// TwinCAT 3 PLC project Main_PLC_Project
// ProgramVersion: 3.1.4023.0
// libraries:
//   Tc2_ControllerToolbox, * (Beckhoff Automation GmbH)
//   Tc2_MC2, * (Beckhoff Automation GmbH)
//   Tc2_MC2_Drive, * (Beckhoff Automation GmbH)
//   Tc2_SerialCom, * (Beckhoff Automation GmbH)
//   Tc2_Standard, * (Beckhoff Automation GmbH)
//   Tc2_System, * (Beckhoff Automation GmbH)
//   Tc3_Filter, * (Beckhoff Automation GmbH)
//   Tc3_Module, * (Beckhoff Automation GmbH)
//   TcMatrix,1.3.0,Burks Engineering
// project tree:
//   DUTs/ E_RobotMode.TcDUT, ST_FilterParams.TcDUT, tDataFrame.TcDUT
//   GVLs/ CONSTANTS.TcGVL, Control.TcGVL, HmiToPlc.TcGVL, Parameters.TcGVL, PlcToHmi.TcGVL, RobotParams.TcGVL, Safety.TcGVL
//   IMU/DUTs/ E_FilterOrder.TcDUT, E_SerialError.TcDUT, E_SerialState.TcDUT, ST_ImuData.TcDUT, ST_JointLimits.TcDUT, ST_JointOffsets.TcDUT, ST_JointParameters.TcDUT, ST_Vector3.TcDUT, tDataFrame_1.TcDUT
//   IMU/GVLs/ IMU.TcGVL
//   IMU/POUs/ ATAN2.TcPOU, BackgroundCOM.TcPOU, FB_AccelerometerAngle.TcPOU, FB_ComplementaryFilter.TcPOU, FB_GetSerialData.TcPOU, FB_MapStim300.TcPOU
//   MATRIX/ AccelerometerReadings.TcPOU, FB_Matrix3x3.TcPOU, FB_Matrix4x4.TcPOU, FB_Vector3.TcPOU, F_Cross2.TcPOU, F_DH.TcPOU
//   / PlcTask.TcTTO, SerialComTask.TcTTO
//   POUs/ FB_Joint.TcPOU, FB_Robot3R.TcPOU, FB_LowPassFilter.TcPOU, FB_TorqueController.TcPOU, FB_TrajectoryGenerator.TcPOU, F_Merge24BitSigned.TcPOU, F_Merge24BitUnsigned.TcPOU, MAIN.TcPOU, P_HMI.TcPOU, RescaleRange.TcPOU
// real-time tasks:
//   TASK PlcTask: cycle T#10ms, priority 20, ADS port 350
//   TASK SerialComTask: cycle T#1ms, priority 1, ADS port 351
// motion (NC):
//   TASK Main_NC_Task SAF: cycle T#2ms, priority 4, ADS port 501
//   TASK Main_NC_Task SVB: cycle T#10ms, priority 8, ADS port 511
//   AXIS Axis1_Drive1_Joint1 (id 1)
//     General: UnitName=°
//     Dynamic: AccelerationMaximum=44, DecelerationMaximum=44, Acceleration=229.701756820377, Deceleration=229.701756820377, Jerk=689.10527046113
//     Velo: RefSearch=1.53134504546918, RefSync=1.53134504546918, SlowManual=7.65672522734589, FastManual=45.9403513640753, Fast=153.134504546918, Maximum=153.134504546918
//     OtherSettings: AllowMotionCmdToSlave=true, PulseDistancePos=1, PulseDistanceNeg=1
//     encoder EncType=8
//       EncPara: ScaleFactorNumerator=5.901639, ScaleFactorDenominator=1048576, MaxCount=#xffffffff
//         SoftEndMinControl: Enable=true, Range=-20
//         SoftEndMaxControl: Enable=true, Range=20
//     drive DrvType=9
//       DrvPara: MaxCount=#xffffffff, DriveControlDWord=#x00030000
//         Analog: VeloReferenz=168.44795500161, VeloScale=1.02400649589962, TorqueSetpointScale=10, ScaleFactorActTorque=0.1
//         TimeComp: TaskDelayCycles=1
//     controller CtrType=1
//       CtrPara: PriorControlFactor=1
//         Observer: BandWidth=20
//   AXIS Axis1_Drive2_Joint2 (id 3)
//     General: UnitName=°
//     Dynamic: AccelerationMaximum=76, DecelerationMaximum=76, Acceleration=389.12958984375, Deceleration=389.12958984375, Jerk=1167.38876953125
//     Velo: RefSearch=2.594197265625, RefSync=2.594197265625, SlowManual=12.970986328125, FastManual=77.82591796875, Fast=259.4197265625, Maximum=259.4197265625
//     OtherSettings: AllowMotionCmdToSlave=true, PulseDistancePos=1, PulseDistanceNeg=1
//     encoder EncType=8
//       EncPara: ScaleFactorNumerator=7.2, ScaleFactorDenominator=1048576, MaxCount=#xffffffff
//         SoftEndMinControl: Enable=true, Range=-95
//         SoftEndMaxControl: Enable=true, Range=95
//     drive DrvType=9
//       DrvPara: MaxCount=#xffffffff, DriveControlDWord=#x00030000
//         Analog: VeloReferenz=285.36169921875, VeloScale=1.02400649589962, TorqueSetpointScale=10, ScaleFactorActTorque=0.1
//         TimeComp: TaskDelayCycles=1
//     controller CtrType=1
//       CtrPara: PriorControlFactor=1
//         Observer: BandWidth=20
//   AXIS Axis1_Drive3_Joint3 (id 5)
//     General: UnitName=Degree
//     Dynamic: AccelerationMaximum=865.888117688623, DecelerationMaximum=865.888117688623, Acceleration=865.888, Deceleration=865.888, Jerk=2597.66, OverrideType=4
//     Velo: RefSearch=5.77258745125749, RefSync=5.77258745125749, SlowManual=28.8629372562874, FastManual=173.177623537725, Fast=577.258745125749, Maximum=577.259
//     OtherSettings: AllowMotionCmdToSlave=true, PulseDistancePos=1, PulseDistanceNeg=1
//     encoder EncType=8
//       EncPara: ScaleFactorNumerator=10.285714, ScaleFactorDenominator=1048576, MaxCount=#xffffffff
//         SoftEndMinControl: Enable=true, Range=-95
//         SoftEndMaxControl: Enable=true, Range=95
//     drive DrvType=9
//       DrvPara: MaxCount=#xffffffff, DriveControlDWord=#x00030000
//         Analog: VeloReferenz=634.984619638324, VeloScale=1.02400649589962, TorqueSetpointScale=10, ScaleFactorActTorque=0.1
//         TimeComp: TaskDelayCycles=1
//     controller CtrType=1
//       CtrPara: PriorControlFactor=1
//         PID: PosTv=0.5, PosTd=0.1, VeloTv=0.2, VeloTd=0.08
//         Observer: BandWidth=20
// I/O:
//   DEVICE Device 5 (EtherCAT), AmsNetId 5.72.215.242.6.1
//     Drive1_Joint1 (AX5106-0000-0210) [AX5106-0000-0210 EtherCAT Drive (SoE, 1 Ch.)]
//       Term 10 (AX5805) [AX5805 (Safety Drive Option)]
//         modules: Module 1 (Safety Process Data, 1 axis), Module 2 (Standard Process Data, 1 axis)
//       Term 7 (EL9011) [EL9011 End Terminal]
//     Drive2_Joint2(AX5106-0000-0210) [AX5106-0000-0210 EtherCAT Drive (SoE, 1 Ch.)]
//       Term 11 (AX5805) [AX5805 (Safety Drive Option)]
//         modules: Module 1 (Safety Process Data, 1 axis), Module 2 (Standard Process Data, 1 axis)
//       Term 8 (EL9011) [EL9011 End Terminal]
//     Drive3_Joint3(AX5106-0000-0210) [AX5106-0000-0210 EtherCAT Drive (SoE, 1 Ch.)]
//       Term 12 (AX5805) [AX5805 (Safety Drive Option)]
//         modules: Module 1 (Safety Process Data, 1 axis), Module 2 (Standard Process Data, 1 axis)
//       Term 9 (EL9011) [EL9011 End Terminal]
//     Box 22 (Leica-RT-Output) [Leica RT Output] (disabled)
//   DEVICE Device 1 (EtherCAT), AmsNetId 5.72.215.242.2.1
//     Term 5 (EK1200) [EK1200-5000 EtherCAT Power supply (2A E-Bus)]
//       Term 14 (EL6900) [EL6900, TwinSAFE PLC]
//       Term 15 (EL1904) [EL1904, 4 Ch. Safety Input 24V, TwinSAFE]
//         modules: Module 1 (FSOES)
//       Term 16 (EL6022) [EL6022 Interface 2Ch. (RS422/485)]
//       Term 19 (EL6022) [EL6022 Interface 2Ch. (RS422/485)]
//       Term 9 (EL9011) [EL9011 End Terminal]
// variable links:
//   Device 1 (EtherCAT) <-> Device 1 (EtherCAT)/Term 5 (EK1200)/Term 14 (EL6900)
//     Term 5 (EK1200)/Term 15 (EL1904)/Module 1 (FSOES)/RxPDO/FSOE <-> ConnectionInputs/Message_9 TxPDO
//     Term 5 (EK1200)/Term 15 (EL1904)/Module 1 (FSOES)/TxPDO/FSOE <-> ConnectionOutputs/Message_9 RxPDO
//   Device 1 (EtherCAT) <-> Device 5 (EtherCAT)/Drive1_Joint1 (AX5106-0000-0210)/Term 10 (AX5805)
//     Term 5 (EK1200)/Term 14 (EL6900)/ConnectionOutputs/Message_6 RxPDO <-> Module 1 (Safety Process Data, 1 axis)/Inputs (Statusword)/FSOE
//   Device 5 (EtherCAT) <-> Device 1 (EtherCAT)/Term 5 (EK1200)/Term 14 (EL6900)
//     Drive1_Joint1 (AX5106-0000-0210)/Term 10 (AX5805)/Module 1 (Safety Process Data, 1 axis)/Outputs (Controlword)/FSOE <-> ConnectionInputs/Message_6 TxPDO
//     Drive2_Joint2(AX5106-0000-0210)/Term 11 (AX5805)/Module 1 (Safety Process Data, 1 axis)/Inputs (Statusword)/FSOE <-> ConnectionOutputs/Message_7 RxPDO
//     Drive3_Joint3(AX5106-0000-0210)/Term 12 (AX5805)/Module 1 (Safety Process Data, 1 axis)/Inputs (Statusword)/FSOE <-> ConnectionOutputs/Message_8 RxPDO
//     Drive2_Joint2(AX5106-0000-0210)/Term 11 (AX5805)/Module 1 (Safety Process Data, 1 axis)/Outputs (Controlword)/FSOE <-> ConnectionInputs/Message_7 TxPDO
//     Drive3_Joint3(AX5106-0000-0210)/Term 12 (AX5805)/Module 1 (Safety Process Data, 1 axis)/Outputs (Controlword)/FSOE <-> ConnectionInputs/Message_8 TxPDO
//   Main_NC_Task SAF/Axes/Axis1_Drive1_Joint1 <-> Device 5 (EtherCAT)/Drive1_Joint1 (AX5106-0000-0210)
//     Drive/Inputs/In/nDcOutputTime <-> InfoData/DcOutputShift
//     Drive/Inputs/In/nState1 <-> AT/Drive status word @bit 8
//     Drive/Inputs/In/nState2 <-> AT/Drive status word
//     Drive/Inputs/In/nState4 @bit 1 <-> WcState/InputToggle
//     Drive/Inputs/In/nState4 <-> WcState/WcState
//     Drive/Outputs/Out/nCtrl1 <-> MDT/Master control word @bit 8
//     Drive/Outputs/Out/nDataOut2 <-> MDT/Velocity command value
//     Enc/Inputs/In/nDataIn1 <-> AT/Position feedback 1 value (motor feedback)
//     Enc/Inputs/In/nDcInputTime <-> InfoData/DcInputShift
//     Enc/Inputs/In/nState4 @bit 1 <-> WcState/InputToggle
//     Enc/Inputs/In/nState4 <-> WcState/WcState
//   Main_NC_Task SAF/Axes/Axis1_Drive2_Joint2 <-> Device 5 (EtherCAT)/Drive2_Joint2(AX5106-0000-0210)
//     Drive/Inputs/In/nDcOutputTime <-> InfoData/DcOutputShift
//     Drive/Inputs/In/nState1 <-> AT/Drive status word @bit 8
//     Drive/Inputs/In/nState2 <-> AT/Drive status word
//     Drive/Inputs/In/nState4 @bit 1 <-> WcState/InputToggle
//     Drive/Inputs/In/nState4 <-> WcState/WcState
//     Drive/Outputs/Out/nCtrl1 <-> MDT/Master control word @bit 8
//     Drive/Outputs/Out/nDataOut2 <-> MDT/Velocity command value
//     Enc/Inputs/In/nDataIn1 <-> AT/Position feedback 1 value (motor feedback)
//     Enc/Inputs/In/nDcInputTime <-> InfoData/DcInputShift
//     Enc/Inputs/In/nState4 @bit 1 <-> WcState/InputToggle
//     Enc/Inputs/In/nState4 <-> WcState/WcState
//   Main_NC_Task SAF/Axes/Axis1_Drive3_Joint3 <-> Device 5 (EtherCAT)/Drive3_Joint3(AX5106-0000-0210)
//     Drive/Inputs/In/nDcOutputTime <-> InfoData/DcOutputShift
//     Drive/Inputs/In/nState1 <-> AT/Drive status word @bit 8
//     Drive/Inputs/In/nState2 <-> AT/Drive status word
//     Drive/Inputs/In/nState4 @bit 1 <-> WcState/InputToggle
//     Drive/Inputs/In/nState4 <-> WcState/WcState
//     Drive/Outputs/Out/nCtrl1 <-> MDT/Master control word @bit 8
//     Drive/Outputs/Out/nDataOut2 <-> MDT/Velocity command value
//     Drive/Outputs/Out/nDataOut4[0] <-> MDT/Torque/force command value
//     Enc/Inputs/In/nDataIn1 <-> AT/Position feedback 1 value (motor feedback)
//     Enc/Inputs/In/nDcInputTime <-> InfoData/DcInputShift
//     Enc/Inputs/In/nState4 @bit 1 <-> WcState/InputToggle
//     Enc/Inputs/In/nState4 <-> WcState/WcState
//   Main_PLC_Project/Main_PLC_Project Instance <-> Device 1 (EtherCAT)/Term 5 (EK1200)/Term 14 (EL6900)
//     PlcTask Inputs/Safety.TS_I_Safety_EStopError <-> StandardInputs/Standard Out Var 5
//     PlcTask Inputs/Safety.TS_I_Safety_EStopOK <-> StandardInputs/Standard Out Var 4
//     PlcTask Outputs/Safety.TS_Q_Safety_Drive_Axis_ErrReset <-> StandardOutputs/Standard In Var 11
//     PlcTask Outputs/Safety.TS_Q_Safety_EStopRestart <-> StandardOutputs/Standard In Var 2
//     PlcTask Outputs/Safety.TS_Q_Safety_GroupPort_ErrAck <-> StandardOutputs/Standard In Var 1
//     PlcTask Outputs/Safety.TS_Q_Safety_GroupPort_RunStop <-> StandardOutputs/Standard In Var 3
//   Main_PLC_Project/Main_PLC_Project Instance <-> Device 1 (EtherCAT)/Term 5 (EK1200)/Term 16 (EL6022)
//     SerialComTask Inputs/IMU.fbStim300[0].stIn_EL6022 @bit 16 <-> COM Inputs Channel 1/Data In 0
//     SerialComTask Inputs/IMU.fbStim300[0].stIn_EL6022 @bit 24 <-> COM Inputs Channel 1/Data In 1
//     SerialComTask Inputs/IMU.fbStim300[0].stIn_EL6022 @bit 96 <-> COM Inputs Channel 1/Data In 10
//     SerialComTask Inputs/IMU.fbStim300[0].stIn_EL6022 @bit 104 <-> COM Inputs Channel 1/Data In 11
//     SerialComTask Inputs/IMU.fbStim300[0].stIn_EL6022 @bit 112 <-> COM Inputs Channel 1/Data In 12
//     SerialComTask Inputs/IMU.fbStim300[0].stIn_EL6022 @bit 120 <-> COM Inputs Channel 1/Data In 13
//     SerialComTask Inputs/IMU.fbStim300[0].stIn_EL6022 @bit 128 <-> COM Inputs Channel 1/Data In 14
//     SerialComTask Inputs/IMU.fbStim300[0].stIn_EL6022 @bit 136 <-> COM Inputs Channel 1/Data In 15
//     SerialComTask Inputs/IMU.fbStim300[0].stIn_EL6022 @bit 144 <-> COM Inputs Channel 1/Data In 16
//     SerialComTask Inputs/IMU.fbStim300[0].stIn_EL6022 @bit 152 <-> COM Inputs Channel 1/Data In 17
//     SerialComTask Inputs/IMU.fbStim300[0].stIn_EL6022 @bit 160 <-> COM Inputs Channel 1/Data In 18
//     SerialComTask Inputs/IMU.fbStim300[0].stIn_EL6022 @bit 168 <-> COM Inputs Channel 1/Data In 19
//     SerialComTask Inputs/IMU.fbStim300[0].stIn_EL6022 @bit 32 <-> COM Inputs Channel 1/Data In 2
//     SerialComTask Inputs/IMU.fbStim300[0].stIn_EL6022 @bit 176 <-> COM Inputs Channel 1/Data In 20
//     SerialComTask Inputs/IMU.fbStim300[0].stIn_EL6022 @bit 184 <-> COM Inputs Channel 1/Data In 21
//     SerialComTask Inputs/IMU.fbStim300[0].stIn_EL6022 @bit 40 <-> COM Inputs Channel 1/Data In 3
//     SerialComTask Inputs/IMU.fbStim300[0].stIn_EL6022 @bit 48 <-> COM Inputs Channel 1/Data In 4
//     SerialComTask Inputs/IMU.fbStim300[0].stIn_EL6022 @bit 56 <-> COM Inputs Channel 1/Data In 5
//     SerialComTask Inputs/IMU.fbStim300[0].stIn_EL6022 @bit 64 <-> COM Inputs Channel 1/Data In 6
//     SerialComTask Inputs/IMU.fbStim300[0].stIn_EL6022 @bit 72 <-> COM Inputs Channel 1/Data In 7
//     SerialComTask Inputs/IMU.fbStim300[0].stIn_EL6022 @bit 80 <-> COM Inputs Channel 1/Data In 8
//     SerialComTask Inputs/IMU.fbStim300[0].stIn_EL6022 @bit 88 <-> COM Inputs Channel 1/Data In 9
//     SerialComTask Inputs/IMU.fbStim300[1].stIn_EL6022 @bit 16 <-> COM Inputs Channel 2/Data In 0
//     SerialComTask Inputs/IMU.fbStim300[1].stIn_EL6022 @bit 24 <-> COM Inputs Channel 2/Data In 1
//     SerialComTask Inputs/IMU.fbStim300[1].stIn_EL6022 @bit 96 <-> COM Inputs Channel 2/Data In 10
//     SerialComTask Inputs/IMU.fbStim300[1].stIn_EL6022 @bit 104 <-> COM Inputs Channel 2/Data In 11
//     SerialComTask Inputs/IMU.fbStim300[1].stIn_EL6022 @bit 112 <-> COM Inputs Channel 2/Data In 12
//     SerialComTask Inputs/IMU.fbStim300[1].stIn_EL6022 @bit 120 <-> COM Inputs Channel 2/Data In 13
//     SerialComTask Inputs/IMU.fbStim300[1].stIn_EL6022 @bit 128 <-> COM Inputs Channel 2/Data In 14
//     SerialComTask Inputs/IMU.fbStim300[1].stIn_EL6022 @bit 136 <-> COM Inputs Channel 2/Data In 15
//     SerialComTask Inputs/IMU.fbStim300[1].stIn_EL6022 @bit 144 <-> COM Inputs Channel 2/Data In 16
//     SerialComTask Inputs/IMU.fbStim300[1].stIn_EL6022 @bit 152 <-> COM Inputs Channel 2/Data In 17
//     SerialComTask Inputs/IMU.fbStim300[1].stIn_EL6022 @bit 160 <-> COM Inputs Channel 2/Data In 18
//     SerialComTask Inputs/IMU.fbStim300[1].stIn_EL6022 @bit 168 <-> COM Inputs Channel 2/Data In 19
//     SerialComTask Inputs/IMU.fbStim300[1].stIn_EL6022 @bit 32 <-> COM Inputs Channel 2/Data In 2
//     SerialComTask Inputs/IMU.fbStim300[1].stIn_EL6022 @bit 176 <-> COM Inputs Channel 2/Data In 20
//     SerialComTask Inputs/IMU.fbStim300[1].stIn_EL6022 @bit 184 <-> COM Inputs Channel 2/Data In 21
//     SerialComTask Inputs/IMU.fbStim300[1].stIn_EL6022 @bit 40 <-> COM Inputs Channel 2/Data In 3
//     SerialComTask Inputs/IMU.fbStim300[1].stIn_EL6022 @bit 48 <-> COM Inputs Channel 2/Data In 4
//     SerialComTask Inputs/IMU.fbStim300[1].stIn_EL6022 @bit 56 <-> COM Inputs Channel 2/Data In 5
//     SerialComTask Inputs/IMU.fbStim300[1].stIn_EL6022 @bit 64 <-> COM Inputs Channel 2/Data In 6
//     SerialComTask Inputs/IMU.fbStim300[1].stIn_EL6022 @bit 72 <-> COM Inputs Channel 2/Data In 7
//     SerialComTask Inputs/IMU.fbStim300[1].stIn_EL6022 @bit 80 <-> COM Inputs Channel 2/Data In 8
//     SerialComTask Inputs/IMU.fbStim300[1].stIn_EL6022 @bit 88 <-> COM Inputs Channel 2/Data In 9
//     SerialComTask Inputs/IMU.fbStim300[0].stIn_EL6022 <-> COM Inputs Channel 1/Status
//     SerialComTask Inputs/IMU.fbStim300[1].stIn_EL6022 <-> COM Inputs Channel 2/Status
//     SerialComTask Outputs/IMU.fbStim300[0].stOut_EL6022 <-> COM Outputs Channel 1/Ctrl
//     SerialComTask Outputs/IMU.fbStim300[1].stOut_EL6022 <-> COM Outputs Channel 2/Ctrl
//     SerialComTask Outputs/IMU.fbStim300[0].stOut_EL6022 @bit 16 <-> COM Outputs Channel 1/Data Out 0
//     SerialComTask Outputs/IMU.fbStim300[0].stOut_EL6022 @bit 24 <-> COM Outputs Channel 1/Data Out 1
//     SerialComTask Outputs/IMU.fbStim300[0].stOut_EL6022 @bit 96 <-> COM Outputs Channel 1/Data Out 10
//     SerialComTask Outputs/IMU.fbStim300[0].stOut_EL6022 @bit 104 <-> COM Outputs Channel 1/Data Out 11
//     SerialComTask Outputs/IMU.fbStim300[0].stOut_EL6022 @bit 112 <-> COM Outputs Channel 1/Data Out 12
//     SerialComTask Outputs/IMU.fbStim300[0].stOut_EL6022 @bit 120 <-> COM Outputs Channel 1/Data Out 13
//     SerialComTask Outputs/IMU.fbStim300[0].stOut_EL6022 @bit 128 <-> COM Outputs Channel 1/Data Out 14
//     SerialComTask Outputs/IMU.fbStim300[0].stOut_EL6022 @bit 136 <-> COM Outputs Channel 1/Data Out 15
//     SerialComTask Outputs/IMU.fbStim300[0].stOut_EL6022 @bit 144 <-> COM Outputs Channel 1/Data Out 16
//     SerialComTask Outputs/IMU.fbStim300[0].stOut_EL6022 @bit 152 <-> COM Outputs Channel 1/Data Out 17
//     SerialComTask Outputs/IMU.fbStim300[0].stOut_EL6022 @bit 160 <-> COM Outputs Channel 1/Data Out 18
//     SerialComTask Outputs/IMU.fbStim300[0].stOut_EL6022 @bit 168 <-> COM Outputs Channel 1/Data Out 19
//     SerialComTask Outputs/IMU.fbStim300[0].stOut_EL6022 @bit 32 <-> COM Outputs Channel 1/Data Out 2
//     SerialComTask Outputs/IMU.fbStim300[0].stOut_EL6022 @bit 176 <-> COM Outputs Channel 1/Data Out 20
//     SerialComTask Outputs/IMU.fbStim300[0].stOut_EL6022 @bit 184 <-> COM Outputs Channel 1/Data Out 21
//     SerialComTask Outputs/IMU.fbStim300[0].stOut_EL6022 @bit 40 <-> COM Outputs Channel 1/Data Out 3
//     SerialComTask Outputs/IMU.fbStim300[0].stOut_EL6022 @bit 48 <-> COM Outputs Channel 1/Data Out 4
//     SerialComTask Outputs/IMU.fbStim300[0].stOut_EL6022 @bit 56 <-> COM Outputs Channel 1/Data Out 5
//     SerialComTask Outputs/IMU.fbStim300[0].stOut_EL6022 @bit 64 <-> COM Outputs Channel 1/Data Out 6
//     SerialComTask Outputs/IMU.fbStim300[0].stOut_EL6022 @bit 72 <-> COM Outputs Channel 1/Data Out 7
//     SerialComTask Outputs/IMU.fbStim300[0].stOut_EL6022 @bit 80 <-> COM Outputs Channel 1/Data Out 8
//     SerialComTask Outputs/IMU.fbStim300[0].stOut_EL6022 @bit 88 <-> COM Outputs Channel 1/Data Out 9
//     SerialComTask Outputs/IMU.fbStim300[1].stOut_EL6022 @bit 16 <-> COM Outputs Channel 2/Data Out 0
//     SerialComTask Outputs/IMU.fbStim300[1].stOut_EL6022 @bit 24 <-> COM Outputs Channel 2/Data Out 1
//     SerialComTask Outputs/IMU.fbStim300[1].stOut_EL6022 @bit 96 <-> COM Outputs Channel 2/Data Out 10
//     SerialComTask Outputs/IMU.fbStim300[1].stOut_EL6022 @bit 104 <-> COM Outputs Channel 2/Data Out 11
//     SerialComTask Outputs/IMU.fbStim300[1].stOut_EL6022 @bit 112 <-> COM Outputs Channel 2/Data Out 12
//     SerialComTask Outputs/IMU.fbStim300[1].stOut_EL6022 @bit 120 <-> COM Outputs Channel 2/Data Out 13
//     SerialComTask Outputs/IMU.fbStim300[1].stOut_EL6022 @bit 128 <-> COM Outputs Channel 2/Data Out 14
//     SerialComTask Outputs/IMU.fbStim300[1].stOut_EL6022 @bit 136 <-> COM Outputs Channel 2/Data Out 15
//     SerialComTask Outputs/IMU.fbStim300[1].stOut_EL6022 @bit 144 <-> COM Outputs Channel 2/Data Out 16
//     SerialComTask Outputs/IMU.fbStim300[1].stOut_EL6022 @bit 152 <-> COM Outputs Channel 2/Data Out 17
//     SerialComTask Outputs/IMU.fbStim300[1].stOut_EL6022 @bit 160 <-> COM Outputs Channel 2/Data Out 18
//     SerialComTask Outputs/IMU.fbStim300[1].stOut_EL6022 @bit 168 <-> COM Outputs Channel 2/Data Out 19
//     SerialComTask Outputs/IMU.fbStim300[1].stOut_EL6022 @bit 32 <-> COM Outputs Channel 2/Data Out 2
//     SerialComTask Outputs/IMU.fbStim300[1].stOut_EL6022 @bit 176 <-> COM Outputs Channel 2/Data Out 20
//     SerialComTask Outputs/IMU.fbStim300[1].stOut_EL6022 @bit 184 <-> COM Outputs Channel 2/Data Out 21
//     SerialComTask Outputs/IMU.fbStim300[1].stOut_EL6022 @bit 40 <-> COM Outputs Channel 2/Data Out 3
//     SerialComTask Outputs/IMU.fbStim300[1].stOut_EL6022 @bit 48 <-> COM Outputs Channel 2/Data Out 4
//     SerialComTask Outputs/IMU.fbStim300[1].stOut_EL6022 @bit 56 <-> COM Outputs Channel 2/Data Out 5
//     SerialComTask Outputs/IMU.fbStim300[1].stOut_EL6022 @bit 64 <-> COM Outputs Channel 2/Data Out 6
//     SerialComTask Outputs/IMU.fbStim300[1].stOut_EL6022 @bit 72 <-> COM Outputs Channel 2/Data Out 7
//     SerialComTask Outputs/IMU.fbStim300[1].stOut_EL6022 @bit 80 <-> COM Outputs Channel 2/Data Out 8
//     SerialComTask Outputs/IMU.fbStim300[1].stOut_EL6022 @bit 88 <-> COM Outputs Channel 2/Data Out 9
//   Main_PLC_Project/Main_PLC_Project Instance <-> Device 1 (EtherCAT)/Term 5 (EK1200)/Term 19 (EL6022)
//     SerialComTask Inputs/IMU.fbStim300[2].stIn_EL6022 @bit {16..184 step 8} <-> COM Inputs Channel 1/Data In {0..21}  (22 links)
//     SerialComTask Inputs/IMU.fbStim300[2].stIn_EL6022 <-> COM Inputs Channel 1/Status
//     SerialComTask Outputs/IMU.fbStim300[2].stOut_EL6022 <-> COM Outputs Channel 1/Ctrl
//     SerialComTask Outputs/IMU.fbStim300[2].stOut_EL6022 @bit {16..184 step 8} <-> COM Outputs Channel 1/Data Out {0..21}  (22 links)
//   Main_PLC_Project/Main_PLC_Project Instance <-> Device 5 (EtherCAT)/Box 22 (Leica-RT-Output)
//     PlcTask Inputs/MAIN.fLeicaRawD <-> Cyclic Measurements/Distance
//     PlcTask Inputs/MAIN.fLeicaRawH <-> Cyclic Measurements/AngleHz
//     PlcTask Inputs/MAIN.fLeicaRawV <-> Cyclic Measurements/AngleVt
//   Main_PLC_Project/Main_PLC_Project Instance <-> Device 5 (EtherCAT)/Drive3_Joint3(AX5106-0000-0210)
//     PlcTask Inputs/MAIN.robot.joints[2].fbTorqueControl.fTorqueFbkPerc <-> AT/Torque/force feedback value
//     PlcTask Inputs/MAIN.robot.joints[2].nVelocityControllerOutputTorque <-> AT/Velocity controller output
//     PlcTask Outputs/MAIN.robot.joints[2].nAdditiveTorquePerc <-> MDT/Additive torque/force command value
//     PlcTask Outputs/MAIN.robot.joints[2].nAdditiveVelocity <-> MDT/Additive velocity command value
//   Main_PLC_Project/Main_PLC_Project Instance <-> Main_NC_Task SAF/Axes/Axis1_Drive1_Joint1
//     PlcTask Inputs/MAIN.robot.joints[0].axis.NcToPlc <-> Outputs/ToPlc
//     PlcTask Outputs/MAIN.robot.joints[0].axis.PlcToNc <-> Inputs/FromPlc
//   Main_PLC_Project/Main_PLC_Project Instance <-> Main_NC_Task SAF/Axes/Axis1_Drive2_Joint2
//     PlcTask Inputs/MAIN.robot.joints[1].axis.NcToPlc <-> Outputs/ToPlc
//     PlcTask Outputs/MAIN.robot.joints[1].axis.PlcToNc <-> Inputs/FromPlc
//   Main_PLC_Project/Main_PLC_Project Instance <-> Main_NC_Task SAF/Axes/Axis1_Drive3_Joint3
//     PlcTask Inputs/MAIN.robot.joints[2].axis.NcToPlc <-> Outputs/ToPlc
//     PlcTask Outputs/MAIN.robot.joints[2].axis.PlcToNc <-> Inputs/FromPlc

CONFIGURATION Main_PLC_Project
    RESOURCE PLC ON TwinCAT3
        TASK PlcTask(INTERVAL := T#10ms, PRIORITY := 20);
        TASK SerialComTask(INTERVAL := T#1ms, PRIORITY := 1);
        PROGRAM MAIN WITH PlcTask : MAIN;
        PROGRAM BackgroundCOM WITH SerialComTask : BackgroundCOM;
    END_RESOURCE
END_CONFIGURATION

// ---- DUTs/E_RobotMode.TcDUT
{attribute 'qualified_only'}
//{attribute 'strict'}
TYPE E_RobotMode : 
(
	NONE := 0,
	ESTOP,
	STOP,
	POSITION,
	VELOCITY,
	TORQUE
)INT;
END_TYPE

// ---- DUTs/ST_FilterParams.TcDUT
TYPE ST_FilterParams :
STRUCT
	// Order
	eOrder 			: E_FilterOrder := E_FilterOrder.eFirst;
	// Cutoff frequency [Hz]
	fCutoff 		: LREAL;
	// Damping ratio [-] (default 0.7071) (Not used in first order)
	fDampingRatio 	: LREAL := SQRT(0.5);
	// Delta time [s]
	fDeltaTime 		: LREAL;
	// Initial value (default 0)
	fInitialValue 	: LREAL := 0.0;
END_STRUCT
END_TYPE

// ---- DUTs/tDataFrame.TcDUT
TYPE tDataFrame :
ARRAY[0..64] OF BYTE; // Normal Mode datagram
END_TYPE

// ---- IMU/DUTs/E_FilterOrder.TcDUT
{attribute 'qualified_only'}
// {attribute 'strict'}
TYPE E_FilterOrder :
(
	eFirst := 0,
	eSecond
);
END_TYPE

// ---- IMU/DUTs/E_SerialError.TcDUT
{attribute 'qualified_only'}
TYPE E_SerialError :
(
	eNoError := 0,
	eComBufferError,
	eOutputBufferTooSmall,
	eChecksumFailed
);
END_TYPE

// ---- IMU/DUTs/E_SerialState.TcDUT
{attribute 'qualified_only'}
TYPE E_SerialState :
(
	eStopped := 0,
	eSearchForHeader,
	eReceive
);
END_TYPE

// ---- IMU/DUTs/ST_ImuData.TcDUT
TYPE ST_ImuData :
STRUCT
	stGyro 	: ST_Vector3;
	stAcc 	: ST_Vector3;
	fRoll 	: LREAL;
	fPitch	: LREAL;
END_STRUCT
END_TYPE

// ---- IMU/DUTs/ST_JointLimits.TcDUT
TYPE ST_JointLimits :
STRUCT
	fMin : LREAL;
	fMax : LREAL;
END_STRUCT
END_TYPE

// ---- IMU/DUTs/ST_JointOffsets.TcDUT
TYPE ST_JointOffsets :
STRUCT
	fPositionOffset 	: LREAL;
	fCalibrationOffset 	: LREAL;
END_STRUCT
END_TYPE

// ---- IMU/DUTs/ST_JointParameters.TcDUT
TYPE ST_JointParameters :
STRUCT
	stOffsets 				: ST_JointOffsets;
	stPositionLimits 		: ST_JointLimits;
	stVelocityLimits 		: ST_JointLimits;
	stAccelerationLimits 	: ST_JointLimits;
END_STRUCT
END_TYPE

// ---- IMU/DUTs/ST_Vector3.TcDUT
TYPE ST_Vector3 :
STRUCT
	x : LREAL;
	y : LREAL;
	z : LREAL;
END_STRUCT
END_TYPE

// ---- IMU/DUTs/tDataFrame_1.TcDUT
TYPE tDataFrame_1 :
ARRAY[0..64] OF BYTE; // Normal Mode datagram
END_TYPE

// ---- GVLs/CONSTANTS.TcGVL
{attribute 'qualified_only'}
VAR_GLOBAL CONSTANT
	DEG_TO_RAD : LREAL := PI/180.0;
	RAD_TO_DEG : LREAL := 180.0/PI;
	GRAVITY : LREAL := 9.81;
	GEAR_RATIO : ARRAY [0..2] OF LREAL := [61.0, 50.0, 35.0];
	TORQUE_SCALING : ARRAY [0..2] OF LREAL := [30.84, 17.21, 2.99]; //converts Nm --> one-tenth of a per cent (‰)  in motor side
	VELOCITY_SCALING : LREAL := EXPT(2.0,30.0)/(360.0*1000.0); //converts deg/s --> rev/2^30 ms  in motor side
END_VAR

// ---- GVLs/Control.TcGVL
{attribute 'qualified_only'}
VAR_GLOBAL

	
END_VAR

// ---- GVLs/HmiToPlc.TcGVL
{attribute 'qualified_only'}
VAR_GLOBAL	
	bEnable : BOOL := FALSE;	
	bReset : BOOL := FALSE;
	bSoftStop : BOOL := FALSE;
	
	
	bSafety_GroupPort_ErrAck : BOOL := FALSE;
	bSafety_EStopRestart  : BOOL := FALSE;	
	bSafety_Drive_Axis_ErrReset : BOOL := FALSE;
	

	fPosInput : ARRAY [0..2] OF LREAL := [90,0,0];
	fVelInput : ARRAY [0..2] OF LREAL := [0,0,0];
	
	eRobotMode : E_RobotMode := E_RobotMode.NONE;
	
	bPositionModeExecute : BOOL := FALSE;
	
	bEnableManualControl : BOOL := FALSE;
	
	bPositionMode : BOOL := FALSE;
	bVelocityMode : BOOL := FALSE;
	bTorqueMode : BOOL := FALSE;
END_VAR

// ---- GVLs/Parameters.TcGVL
{attribute 'qualified_only'}
VAR_GLOBAL PERSISTENT
//	fJointPositionOffset 	: ARRAY [0..2] OF LREAL := [ 90.0, 0.0, 0.0 ];
//	fJointCalibrationOffset : ARRAY [0..2] OF LREAL := [ -0.145, 1.69, -1.54 ];
//	fJointLimitsMin : ARRAY [0..2] OF LREAL := [ 75.0, -90.0, -90.0 ]; //in robot coordinates
//	fJointLimitsMax : ARRAY [0..2] OF LREAL := [ 105.0, 90.0, 90.0 ]; //in robot coordinates
	stJointParams : ARRAY [0..2] OF ST_JointParameters := [
		(	
			stOffsets 				:= (
				fPositionOffset 	:= 90.0,
			    fCalibrationOffset  := -0.145
			),
			stPositionLimits 		:= (
				fMin := 75.0,
				fMax := 105.0
			),
			stVelocityLimits 		:= (
				fMin := 0.0,
				fMax := 0.0
			),
			stAccelerationLimits 	:= (
				fMin := 0.0,
				fMax := 0.0
			)

		),
		(	
			stOffsets 				:= (
				fPositionOffset 	:= 0.0,
			    fCalibrationOffset  := 1.69
			),
			stPositionLimits 		:= (
				fMin := -90.0,
				fMax := 90.0
			),
			stVelocityLimits 		:= (
				fMin := 0.0,
				fMax := 0.0
			),
			stAccelerationLimits 	:= (
				fMin := 0.0,
				fMax := 0.0
			)

		),
		(	
			stOffsets 				:= (
				fPositionOffset 	:= 0.0,
			    fCalibrationOffset  := -1.54
			),
			stPositionLimits 		:= (
				fMin := -90.0,
				fMax := 90.0
			),
			stVelocityLimits 		:= (
				fMin := 0.0,
				fMax := 0.0
			),
			stAccelerationLimits 	:= (
				fMin := 0.0,
				fMax := 0.0
			)

		)
	];
END_VAR

// ---- GVLs/PlcToHmi.TcGVL
{attribute 'qualified_only'}
VAR_GLOBAL
	
	fPosFb  : ARRAY [0..2] OF LREAL;
	fVelFb  : ARRAY [0..2] OF LREAL;
	fTauFb 	: ARRAY [0..2] OF LREAL;
	
	bPositionMode 	: BOOL;
	bVelocityMode 	: BOOL;
	bTorqueMode 	: BOOL;
	
	bSafety_EStopOK  : BOOL;
	bSafety_EStopError : BOOL;
	
	bAnyJointActive : BOOL;
END_VAR

// ---- GVLs/RobotParams.TcGVL
{attribute 'qualified_only'}
VAR_GLOBAL
	fLinkLength : ARRAY [0..2] OF LREAL := [1.5, 1.5, 1.5];
	fLinkMass : ARRAY [0..2] OF LREAL := [2.9809, 1.7982, 1.1138];
	fHubMass : ARRAY [0..2] OF LREAL := [51.2960, 12.4690, 4.2810];
	fPayloadMass : LREAL := 0.0;
	fGravity : LREAL := 9.81;
END_VAR

// ---- GVLs/Safety.TcGVL
{attribute 'qualified_only'}
VAR_GLOBAL
	TS_Q_Safety_GroupPort_ErrAck AT %Q* : BOOL;
	TS_Q_Safety_EStopRestart AT %Q* : BOOL;
	TS_Q_Safety_GroupPort_RunStop AT %Q* : BOOL := TRUE;
	
	TS_Q_Safety_Drive_Axis_ErrReset AT %Q* : BOOL;
		
	TS_I_Safety_EStopOK AT %I* : BOOL;
	TS_I_Safety_EStopError AT %I* : BOOL;
	
END_VAR

// ---- IMU/GVLs/IMU.TcGVL
{attribute 'qualified_only'}
{attribute 'TcContextName':='SerialComTask'} //the variables in this lib are sync with the SerialComTask
VAR_GLOBAL
	fbStim300 : ARRAY [0..2] OF FB_MapStim300;	
END_VAR

// ---- POUs/MAIN.TcPOU
PROGRAM MAIN
VAR_INPUT
	robot : FB_Robot3R;
	fPosInput : ARRAY [0..2] OF LREAL;
	fVelInput : ARRAY [0..2] OF LREAL;	
END_VAR
VAR
	bDelayStart : BOOL := FALSE;
	fbDelayStart : TON := (PT := T#2S);
	
	
	
//	t AT %Q* : LREAL;
//	A : ARRAY [0..2] OF LREAL;
//	w : ARRAY [0..2] OF LREAL;
//	TT : ARRAY [0..2] OF LREAL;
//	q_Offset : ARRAY [0..2] OF LREAL;
//	phi_Offset : ARRAY [0..2] OF LREAL;
//	y : ARRAY [0..2] OF LREAL;
//	y_t : ARRAY [0..2] OF LREAL;
	u : ARRAY [0..2] OF LREAL;
	
	j : USINT;
//	i : USINT;
	
	
	timers : ARRAY [0..3] OF TON;
	
	// Task cycle time monitoring
	Ts : LREAL := 0.01;
	fbGetCurrentTaskIdx : GETCURTASKINDEX;
	bCycleTimeExceeded : BOOL;
	nCycleCount : UDINT;

	
	bEStop : BOOL;
	
	bRunStupidRoutine: BOOL;
	
	bVelocityMode : BOOL;
	bPositionMode : BOOL;
	bStop : BOOL;
	
	// IK Data
//	Vt AT %Q* : LREAL := 0.5;
//	radius AT %Q* : LREAL := 0.5;
//	p0 AT %Q* : ARRAY [0..1] OF LREAL := [1.5, 2.5];
//	L  AT %Q* : ARRAY [0..2] OF LREAL := [1.5, 1.5, 1.5];

//	q_t  AT %I* : ARRAY [0..2] OF LREAL;
//	q  AT %I* : ARRAY [0..2] OF LREAL;
	
	
	
//	q_t_DEG : ARRAY [0..2] OF LREAL;
//	q_DEG : ARRAY [0..2] OF LREAL;
	
	deflection : ARRAY [0..2] OF LREAL;
	cumulativeAngle : ARRAY [0..2] OF LREAL;
//	cumulativeVel : LREAL;



	// Calculate deflection using new approach
	deflectionNew : ARRAY [0..2] OF LREAL;
	
	//filters
	fbGyroFilters : ARRAY [0..2] OF FB_LowPassFilter;
	fGyroFilterCutoff : ARRAY [0..2] OF LREAL := [ 10.0, 10.0, 10.0 ];
	fLinkGyroVelocity : ARRAY [0..2] OF LREAL;
	stGyroFilterParams : ST_FilterParams;
	bFirstRun : BOOL := TRUE;
	
	// Additive torque based on deflection measurement	
	fShaftAdditiveTorque : ARRAY [0..2] OF LREAL := [0.0, 0.0, 0.0]; // [Nm]
	Kt : ARRAY [0..2] OF LREAL := [0.0, 0.0, 0.0]; // gain for defelectuib compensation
	bEnableDeflectionCompensation : BOOL := FALSE;
	
	// Additive velocity based on deflection measurement	
	fShaftAdditiveVelocity : ARRAY [0..2] OF LREAL := [0.0, 0.0, 0.0]; // [Nm]
	
	//filters for velocity feeback
	fbJointVelFilters : ARRAY [0..2] OF FB_LowPassFilter;
	fJointVelFilterCutoff : ARRAY [0..2] OF LREAL := [ 10.0, 10.0, 10.0 ];
	
	q_t_Filtered : ARRAY [0..2] OF LREAL;
	stJointVelFilterParams : ST_FilterParams;
	
	fElasticOscilationVelocity : ARRAY [0..2] OF LREAL;//differene between joint veocity and velocity measured by gyro
	fElasticOscilationVelocityFiltered : ARRAY [0..2] OF LREAL;//differene between joint veocity and velocity measured by gyro
	fElasticOscilationVelocityLast : ARRAY [0..2] OF LREAL := [0.0, 0.0, 0.0];

	fElasticOscilationAcceleration : ARRAY [0..2] OF LREAL;// d(Vel)/dt
	fElasticOscilationVeloHighPass : ARRAY [0..2] OF LREAL;
	
	//filters for link oscillations feeback
	fbElasticOscilationVelocityFilters : ARRAY [0..2] OF FB_LowPassFilter;
	stElasticOscilationVelocityFilterParams : ARRAY [0..2] OF ST_FilterParams := [
		(	
			eOrder := E_FilterOrder.eSecond,
			fCutoff := 10
		),
		(
			eOrder := E_FilterOrder.eSecond,
			fCutoff := 10
		),
		(
			eOrder := E_FilterOrder.eSecond,
			fCutoff := 10
		)
	];
	
//	nVelocityFeedbackRaw AT %I* : DINT;
//	fVelocityFeedback : LREAL;


//	// implement integrator
//	fVibrationFeedback : ARRAY [0..2] OF LREAL := [0.0, 0.0, 0.0];
//	Kf : ARRAY [0..2] OF LREAL := [0.0, 0.0, 0.0]; // gain for defelectuib compensation
//	fIntegrand : ARRAY [0..2] OF LREAL := [0.0, 0.0, 0.0];
//	fIntegOut : ARRAY [0..2] OF LREAL := [0.0, 0.0, 0.0];
//	fCompOut : ARRAY [0..2] OF LREAL := [0.0, 0.0, 0.0];


//	// implement high pass filtering on deflection
//filters for link oscillations feeback
	fbDeflectionFilters : ARRAY [0..2] OF FB_LowPassFilter;
	stDeflectionFilterParams : ARRAY [0..2] OF ST_FilterParams := [
		(	
			eOrder := E_FilterOrder.eSecond,
			fCutoff := 1
		),
		(
			eOrder := E_FilterOrder.eSecond,
			fCutoff := 1
		),
		(
			eOrder := E_FilterOrder.eSecond,
			fCutoff := 1
		)
	];
	fDeflectionHighPass : ARRAY [0..2] OF LREAL;
	fDeflectionLowPassFiltered : ARRAY [0..2] OF LREAL;
	
	//// Calculate deflection using new approach: filters----------------------------------------
	fbDeflectionNewFilters : ARRAY [0..2] OF FB_LowPassFilter;
	fDeflectionNewHighPass : ARRAY [0..2] OF LREAL;
	fDeflectionNewLowPassFiltered : ARRAY [0..2] OF LREAL;//-----------------------------------------
	
	fKf : ARRAY [0..2] OF LREAL := [0.0, 0.0, 0.0]; // gain for defelectuib compensation
	fShaftAdditiveVelocityTest : ARRAY [0..2] OF LREAL := [0.0, 0.0, 0.0]; 
	
	fCalibrationOffset : ARRAY [0..2] OF LREAL;
	
	
	
	
	//joint acceleration low pass filters
	fbJointAccFilters : ARRAY [0..2] OF FB_LowPassFilter;
	stJointAccFilterParams : ARRAY [0..2] OF ST_FilterParams := [
		(	
			eOrder := E_FilterOrder.eSecond,
			fCutoff := 50
		),
		(
			eOrder := E_FilterOrder.eSecond,
			fCutoff := 50
		),
		(
			eOrder := E_FilterOrder.eSecond,
			fCutoff := 50
		)
	];
	fJointAccLowPassFiltered : ARRAY [0..2] OF LREAL;
	
	//Leica Readings
	fLeicaRawH AT %I*: LREAL; //rad
	fLeicaRawV AT %I*: LREAL; //rad
	fLeicaRawD AT %I*: LREAL; //m
	
	
	//Leica Readings
	fXLeica : LREAL := 0.0; //m
	fYLeica : LREAL := 0.0; //m
	fZLeica : LREAL := 0.0; //m
		

	//Accelerometer Readings Compensation
	q_rad : ARRAY [0..2] OF LREAL;
	qdot_rad : ARRAY [0..2] OF LREAL;
	qddot_rad : ARRAY [0..2] OF LREAL;
	
	AccelerometerReadingsOut : ARRAY [0..2] OF FB_Vector3;	
	Tip_to_IMU : ARRAY [0..2] OF FB_Vector3;
	L : ARRAY [0..2] OF LREAL := [1.5,1.5,1.5];
	gravity_vector : FB_Vector3 := (X := 0, Y := 9.81, Z := 0);
	
	
	
	
END_VAR

IF bDelayStart THEN
	fbDelayStart(IN := TRUE);
	IF fbDelayStart.Q THEN
		fbDelayStart(IN := FALSE);
		bDelayStart := FALSE;
	END_IF
	RETURN;
END_IF

P_HMI();

stupidRoutine(bRunStupidRoutine:=bRunStupidRoutine);


// Get smaple time from current task
getSampleTime();


IF bFirstRun THEN
	bFirstRun := FALSE;
	FOR j := 0 TO 2 DO
		//initialize Gyro Filters
		stGyroFilterParams.fCutoff := fGyroFilterCutoff[j];
		stGyroFilterParams.fDeltaTime := Ts;
		stGyroFilterParams.fInitialValue := 0.0;
		fbGyroFilters[j].init(stParams := stGyroFilterParams);
		
		//initialize JointVel Filters
		stJointVelFilterParams.fCutoff := fJointVelFilterCutoff[j];
		stJointVelFilterParams.fDeltaTime := Ts;
		stJointVelFilterParams.fInitialValue := 0.0;
		fbJointVelFilters[j].init(stParams := stJointVelFilterParams);
		
		// filters for link oscillations feeback
		stElasticOscilationVelocityFilterParams[j].fDeltaTime := Ts;
		fbElasticOscilationVelocityFilters[j].init(stParams := stElasticOscilationVelocityFilterParams[j]);
		
		//filters for deflection
		stDeflectionFilterParams[j].fDeltaTime := Ts;
		fbDeflectionFilters[j].init(stParams := stDeflectionFilterParams[j]);
		
		
		//filters for deflectionNew
		fbDeflectionNewFilters[j].init(stParams := stDeflectionFilterParams[j]);
		
		//filter for joint acc
		stJointAccFilterParams[j].fDeltaTime := Ts;
		fbJointAccFilters[j].init(stParams := stJointAccFilterParams[j]);
		
	END_FOR
END_IF





// cumulativeAngle[0] := robot.q[0];
//cumulativeVel := 0.0;
FOR j := 0 TO 2 DO
	fbGyroFilters[j].update(IMU.fbStim300[j].ImuData.stGyro.x);
	fLinkGyroVelocity[j] := fbGyroFilters[j].fOut;
	IF j > 0 THEN
		fLinkGyroVelocity[j] := fLinkGyroVelocity[j] - fbGyroFilters[j-1].fOut;
		cumulativeAngle[j] := cumulativeAngle[j-1] + robot.q[j];
	ELSE
		cumulativeAngle[j] := robot.q[j];
	END_IF
	
	deflection[j] := IMU.fbStim300[j].fRollDeg - cumulativeAngle[j];
END_FOR



FOR j := 0 TO 2 DO
	IF j > 0 THEN
		deflectionNew[j] := IMU.fbStim300[j].fRollDeg - (robot.q[j] + IMU.fbStim300[j-1].fRollDeg);
	ELSE
		deflectionNew[j] := IMU.fbStim300[j].fRollDeg - robot.q[j];
	END_IF
	
	//high pass filtering on deflection and removing static deflection terms
	fbDeflectionNewFilters[j].update(deflectionNew[j]);
	fDeflectionNewLowPassFiltered[j] := fbDeflectionNewFilters[j].fOut;
	fDeflectionNewHighPass[j] := deflectionNew[j] - fDeflectionNewLowPassFiltered[j];
	
END_FOR




//calculate additive torque
FOR j := 0 TO 2 DO	
	fbJointVelFilters[j].update(robot.q_t[j]);
	q_t_Filtered[j] := fbJointVelFilters[j].fOut;
	fElasticOscilationVelocity[j] := fLinkGyroVelocity[j] - q_t_Filtered[j];
	fElasticOscilationVelocityFiltered[j] := fbElasticOscilationVelocityFilters[j].update(fElasticOscilationVelocity[j]);
	
	fElasticOscilationAcceleration[j] := (fElasticOscilationVelocityFiltered[j] - fElasticOscilationVelocityLast[j])/Ts;
	fElasticOscilationVelocityLast[j] := fElasticOscilationVelocityFiltered[j];
	
	fElasticOscilationVeloHighPass[j] := fElasticOscilationVelocity[j] - fElasticOscilationVelocityFiltered[j];

(*	
//	// integrator
//	fVibrationFeedback[j] := fElasticOscilationVelocityFiltered[j];
//	//
//	fIntegOut[j] := fIntegOut[j] + q_t_Filtered[j]*fVibrationFeedback[j]*Ts;	
//	fCompOut[j] := -Kf[j]*fVibrationFeedback[j]*fIntegOut[j]; //doesnot work and it is very dangerous to integrate
*)

	//high pass filtering on deflection and removing static deflection terms
	fbDeflectionFilters[j].update(deflection[j]);
	fDeflectionLowPassFiltered[j] := fbDeflectionFilters[j].fOut;
	fDeflectionHighPass[j] := deflection[j] - fDeflectionLowPassFiltered[j];
	
	fShaftAdditiveVelocityTest[j] := -fKf[j]*fDeflectionNewHighPass[j];
	
	
	
	
	
	IF bEnableDeflectionCompensation THEN	
//		fShaftAdditiveTorque[j] := -Kt[j]*fElasticOscilationVelocity[j];
//		fShaftAdditiveVelocity[j] := -Kt[j]*fElasticOscilationVelocityFiltered[j];
//		fShaftAdditiveVelocity[j] := -Kt[j]*fElasticOscilationVeloHighPass[j]; //doesnot work
		
		fShaftAdditiveVelocity[j] := fShaftAdditiveVelocityTest[j];

	ELSE
		fShaftAdditiveTorque[j] := 0.0;
		fShaftAdditiveVelocity[j] := 0.0;	
	END_IF		
END_FOR




robot(
	bEmStop := NOT Safety.TS_I_Safety_EStopOK,
	Ts:=Ts,
	fVelInput:=fVelInput,//u
	fPosInput := fPosInput,
	fShaftAdditiveTorque := fShaftAdditiveTorque,
	fShaftAdditiveVelocity := fShaftAdditiveVelocity,
	stJointParams := Parameters.stJointParams,
	fDeflection := fDeflectionNewLowPassFiltered
//	fJointPositionOffset := Parameters.fJointPositionOffset,
//	fJointCalibrationOffset := Parameters.fJointCalibrationOffset
);

//joint acc filtered
FOR j := 0 TO 2 DO
	fbJointAccFilters[j].update(robot.q_tt[j]);
	fJointAccLowPassFiltered[j] := fbJointAccFilters[j].fOut;
END_FOR


//fVelocityFeedback := TO_LREAL(nVelocityFeedbackRaw)/(CONSTANTS.VELOCITY_SCALING*CONSTANTS.GEAR_RATIO[2]);

FOR j := 0 TO 2 DO
	fCalibrationOffset[j] := IMU.fbStim300[j].fRollDegFiltered - robot.q[j];
	IF (j <> 0) THEN
		fCalibrationOffset[j] := fCalibrationOffset[j] - 90;
	END_IF
END_FOR



//Leica Data
fXLeica := fLeicaRawD*SIN(fLeicaRawV)*COS(fLeicaRawH);
fYLeica := fLeicaRawD*SIN(fLeicaRawV)*SIN(fLeicaRawH);
fZLeica := fLeicaRawD*COS(fLeicaRawV);



//Accelerometer Readings Compensation
Tip_to_IMU[0].X := 0;
Tip_to_IMU[0].Y := -0.1;
Tip_to_IMU[0].Z := -0.0198;

Tip_to_IMU[1].X := 0;
Tip_to_IMU[1].Y := -0.1;
Tip_to_IMU[1].Z := -0.0198;

Tip_to_IMU[2].X := 0;
Tip_to_IMU[2].Y := -0.1;
Tip_to_IMU[2].Z := -0.0198;

FOR j := 0 TO 2 DO
	q_rad[j] :=  robot.q[j]*CONSTANTS.DEG_TO_RAD;	
	qdot_rad[j] :=  q_t_Filtered[j]*CONSTANTS.DEG_TO_RAD;	
	qddot_rad[j] :=  fJointAccLowPassFiltered[j]*CONSTANTS.DEG_TO_RAD;	 
END_FOR

AccelerometerReadings(
	q:=q_rad,
	qdot:=qdot_rad,
	qddot:=qddot_rad,
	L:=L,
	Tip_to_IMU:=Tip_to_IMU,
	AccelerometerReadingsOut := AccelerometerReadingsOut,
	gravity_vector := gravity_vector
);

ACTION getSampleTime:
// Get sample time of current task
fbGetCurrentTaskIdx();
bCycleTimeExceeded := _TaskInfo[fbGetCurrentTaskIdx.index].CycleTimeExceeded;
nCycleCount := _TaskInfo[fbGetCurrentTaskIdx.index].CycleCount;
Ts := UDINT_TO_LREAL(_TaskInfo[fbGetCurrentTaskIdx.index].CycleTime/10)/1E6;
END_ACTION

METHOD stupidRoutine : BOOL
VAR_INPUT
	bRunStupidRoutine: BOOL;
END_VAR
timers[0](
	IN:=bRunStupidRoutine,
	PT:=T#2S
);

IF timers[0].Q THEN
	Safety.TS_Q_Safety_GroupPort_ErrAck := TRUE;
	
	timers[1](
		IN:=bRunStupidRoutine,
		PT:=T#1S
	);
	
	IF timers[1].Q THEN
		Safety.TS_Q_Safety_GroupPort_ErrAck := FALSE;
		Safety.TS_Q_Safety_EStopRestart := TRUE;
		
		timers[2](
			IN:=bRunStupidRoutine,
			PT:=T#1S
		);
		
		IF timers[2].Q THEN
			Safety.TS_Q_Safety_EStopRestart := FALSE;
			Safety.TS_Q_Safety_Drive_Axis_ErrReset := TRUE;
			
			timers[3](
				IN:=bRunStupidRoutine,
				PT:=T#1S
			);
			
			IF timers[3].Q THEN
				Safety.TS_Q_Safety_Drive_Axis_ErrReset := FALSE;
				
			END_IF
			
		END_IF
		
	END_IF
	
END_IF
END_METHOD

END_PROGRAM

// ---- POUs/FB_Robot3R.TcPOU
FUNCTION_BLOCK FB_Robot3R
VAR_INPUT
	bEmStop : BOOL;
	Ts : LREAL := 0.01;
	bReset : BOOL;
	bEnable : BOOL;
	bEnableJoint : ARRAY [0..2] OF BOOL;
	eRobotModeCmd : E_RobotMode;
	fVelInput : ARRAY [0..2] OF LREAL;
	fPosInput : ARRAY [0..2] OF LREAL;	
	fShaftAdditiveTorque : ARRAY [0..2] OF LREAL; // [Nm]
	fShaftAdditiveVelocity : ARRAY [0..2] OF LREAL; // [deg/sec]
	bPositionModeExecute 	: BOOL;
	bAddDeflection : BOOL := FALSE;
	fDeflection : ARRAY [0..2] OF LREAL := [0.0,0.0,0.0];
	fDeflectionGain : ARRAY [0..2] OF LREAL := [1.0, 1.0,1.0];
//	fJointPositionOffset 	: ARRAY [0..2] OF LREAL;	
//	fJointCalibrationOffset : ARRAY [0..2] OF LREAL;
//	fJointLimitMin : ARRAY [0..2] OF LREAL;	
//	fJointLimitMax : ARRAY [0..2] OF LREAL;
	stJointParams : ARRAY [0..2] OF ST_JointParameters;
		fPosThreshold : LREAL := 0.005;
END_VAR
VAR_OUTPUT
	eRobotMode : E_RobotMode := E_RobotMode.STOP;
	
	fPosDiff : ARRAY [0..2] OF LREAL;
	fDeflectionCompensation : ARRAY [0..2] OF LREAL;
	
	// Robot feedback
	q : ARRAY [0..2] OF LREAL;
	q_t : ARRAY [0..2] OF LREAL;	
	tau : ARRAY [0..2] OF LREAL;
	//the following two lines is added to remove the joint acc from imu readings
	q_t_old : ARRAY [0..2] OF LREAL := [0.0, 0.0, 0.0];
	q_tt : ARRAY [0..2] OF LREAL;
	
	bAnyJointActive : BOOL;
	// Setpoints
	qRef : ARRAY [0..2] OF LREAL;
	qRef_t : ARRAY [0..2] OF LREAL;
	qRef_tt : ARRAY [0..2] OF LREAL;
END_VAR
VAR

	
	fLimitedPosInput : ARRAY [0..2] OF LREAL;
	
	fShaftTorqueRef : ARRAY [0..2] OF LREAL;

	i : USINT;
	j : USINT;
	k : USINT;
	joints : ARRAY [0..2] OF FB_Joint;
		
	//Velcity of last timestamp
	fVelInputOld : ARRAY [0..2] OF LREAL;
	
	
	//Torque oontrol
	Kp : ARRAY [0..2] OF LREAL := [20, 20, 20];
	Kd : ARRAY [0..2] OF LREAL := [5, 5, 5];
	fGravityTorque : ARRAY [0..2] OF LREAL := [0.0, 0.0, 0.0];//shouldnot be zero
	fbPid : FB_CTRL_PID;
	stPidParams : ST_CTRL_PID_PARAMS;
	ePidMode : E_CTRL_MODE;
	bInitPidControl : BOOL := TRUE;
	
	//filters for velocity feeback
	fbJointVelFilters : ARRAY [0..2] OF FB_LowPassFilter;
	fJointVelFilterCutoff : ARRAY [0..2] OF LREAL := [ 10.0, 10.0, 10.0 ];
	q_t_Filtered : ARRAY [0..2] OF LREAL;
	stJointVelFilterParams : ST_FilterParams;
	bFirstRun : BOOL := TRUE;
	

	//trajectory generation
	fbTrajectoryGenerator : ARRAY [0..2] OF FB_TrajectoryGenerator;
	ft : ARRAY [0..2] OF LREAL := [0.0,0.0,0.0];
	ftf : LREAL := 5.0;
	fPosInputOld : ARRAY [0..2] OF LREAL;	
	bExecuteReady : ARRAY [0..2] OF BOOL := [FALSE, FALSE, FALSE];	
	
	
	
	
	//PD control in position loop
		//Torque oontrol
	KpPos : ARRAY [0..2] OF LREAL := [0.2, 0.2, 0.2];
	KdPos : ARRAY [0..2] OF LREAL := [0.0, 0.0, 0.0];
	KffPos : ARRAY [0..2] OF LREAL := [1, 1, 1];
END_VAR

IF bEmStop AND (eRobotMode <> E_RobotMode.ESTOP) THEN
	eRobotModeCmd := E_RobotMode.ESTOP;
END_IF

IF eRobotModeCmd <> E_RobotMode.NONE THEN
	CASE eRobotModeCmd OF
		 E_RobotMode.STOP:
		 	
			
		 	eRobotMode := E_RobotMode.STOP;
			
		 E_RobotMode.ESTOP:
		 	eRobotMode := E_RobotMode.ESTOP;
		 
		 E_RobotMode.POSITION:
				
		 	eRobotMode := E_RobotMode.POSITION;
		 
		 E_RobotMode.VELOCITY:
		 	
		 	eRobotMode := E_RobotMode.VELOCITY;
			
		E_RobotMode.TORQUE:
			eRobotMode := E_RobotMode.TORQUE;
			
	END_CASE	
END_IF
eRobotModeCmd := E_RobotMode.NONE;

IF bReset AND NOT(bEmStop)  THEN
	eRobotMode := E_RobotMode.STOP;
END_IF

// E-stop mode
IF(eRobotMode = E_RobotMode.ESTOP) THEN
	bEnable := FALSE;
	bReset := TRUE;	//to avoid error: the axis loss the enable signal while doing something
END_IF


bAnyJointActive := joints[0].bActive;
FOR k:= 1 TO 2 DO
	bAnyJointActive := bAnyJointActive OR joints[k].bActive;	
END_FOR

IF(eRobotMode = E_RobotMode.STOP) AND  NOT bAnyJointActive THEN
	bEnable := FALSE;
END_IF

FOR i := 0 TO 2 DO
	fLimitedPosInput[i] := LIMIT(
		stJointParams[i].stPositionLimits.fMin,
		fPosInput[i],
		stJointParams[i].stPositionLimits.fMax
	);	
END_FOR

// position mode
IF(eRobotMode = E_RobotMode.POSITION) THEN
	positionMode();
// velocity mode
ELSIF(eRobotMode = E_RobotMode.VELOCITY) THEN
	velocityMode();
ELSIF(eRobotMode = E_RobotMode.TORQUE) THEN
//	torqueMode(); //calculate ref torque in all modes???
END_IF

torqueMode(); //update referece torque all the time so that we don't receive too high command in the start


// Execute joints
FOR j:= 0 TO 2 DO
	joints[j](
		bReset:=bReset,
		bEnable:=bEnable AND bEnableJoint[j],
		eRobotMode := eRobotMode,
		bPositionModeExecute := bPositionModeExecute,
		fGearRatio := CONSTANTS.GEAR_RATIO[j],
		fTorqueScaling := CONSTANTS.TORQUE_SCALING[j],
		qRef:=qRef[j],
		qRef_t := qRef_t[j],
		qRef_tt:=qRef_tt[j],
		fShaftAdditiveTorque := fShaftAdditiveTorque[j],
		fShaftAdditiveVelocity := fShaftAdditiveVelocity[j],
		fShaftTorqueRef  :=  fShaftTorqueRef[j],
//		fOffset := stJointParams[j].stOffsets.fCalibrationOffset + stJointParams[j].stOffsets.fPositionOffset, // fJointPositionOffset[j] + fJointCalibrationOffset[j],
		stJointParams := stJointParams[j],
		Ts := Ts
	);

	// Assign feedback data from joints
	q[j] := joints[j].q;
	q_t[j] := joints[j].q_t;
	tau[j] := joints[j].tau;
	
	q_tt[j] := (q_t[j] - q_t_old[j])/Ts;
	q_t_old[j] := q_t[j];
		
END_FOR

METHOD PRIVATE positionMode : BOOL
VAR_INPUT
	
END_VAR

FOR i:= 0 TO 2 DO
	IF joints[i].bActive THEN		
		// Set input based on velocity input u
		qRef[i] := fPosInput[i];
		qRef_t[i] := fVelInput[i];
		
	END_IF
	
END_FOR
END_METHOD

METHOD PRIVATE torqueMode : BOOL
VAR_INPUT
END_VAR
IF bInitPidControl THEN
	stPidParams.tCtrlCycleTime := T#10MS;
	stPidParams.tTaskCycleTime := T#10MS;
	stPidParams.fKp := 0.1;
	stPidParams.tTn                    := T#1000MS; 
	stPidParams.tTv                    := T#100MS; 
	stPidParams.tTd                    := T#100MS; 
	stPidParams.fOutMaxLimit           := 20; //Nm
	stPidParams.fOutMinLimit           := -20; //NM
	stPidParams.bPInTheFeedbackPath    := FALSE;
	stPidParams.bDInTheFeedbackPath    := TRUE;
	stPidParams.bARWOnIPartOnly        := FALSE;
	
	ePidMode := eCTRL_MODE_ACTIVE; 
	bInitPidControl := FALSE;
END_IF


fbPid(fSetpointValue := fPosInput[2],
		fActualValue := joints[2].q,
		eMode := ePidMode,
		stParams := stPidParams);


IF bFirstRun THEN
	bFirstRun := FALSE;
	FOR i := 0 TO 2 DO
		
		//initialize JointVel Filters
		stJointVelFilterParams.fCutoff := fJointVelFilterCutoff[i];
		stJointVelFilterParams.fDeltaTime := Ts;
		stJointVelFilterParams.fInitialValue := 0.0;
		fbJointVelFilters[i].init(stParams := stJointVelFilterParams);
		
	END_FOR
END_IF		
		
		
fGravityTorque[2] := (RobotParams.fLinkMass[2]/2.0 + RobotParams.fPayloadMass)*RobotParams.fGravity*RobotParams.fLinkLength[2]*COS((joints[0].q + joints[1].q + joints[2].q)*CONSTANTS.DEG_TO_RAD);



FOR i:= 0 TO 2 DO
//	IF joints[i].bActive THEN		
		// get input position from HMI		
		//calculate gravity torque
		
//		fShaftTorqueRef[i] :=  fbPid.fOut;
		fbJointVelFilters[i].update(joints[i].q_t);
		q_t_Filtered[i] := fbJointVelFilters[i].fOut;
		fShaftTorqueRef[i] := fShaftAdditiveTorque[i] + Kp[i]*(fPosInput[i] - joints[i].q)* CONSTANTS.DEG_TO_RAD + Kd[i]*(0.0 - q_t_Filtered[i])*CONSTANTS.DEG_TO_RAD + fGravityTorque[i]; //add gravity torque here 
		
//	END_IF	
END_FOR
END_METHOD

METHOD PRIVATE velocityMode : BOOL
VAR_INPUT
END_VAR
VAR
	
END_VAR
// Integrate position

FOR i:= 0 TO 2 DO
	IF bAddDeflection THEN
		fDeflectionCompensation[i] :=  fDeflectionGain[i] *fDeflection[i];
	ELSE			
		fDeflectionCompensation[i] := 0.0;
	END_IF
	
//	qRef[i] := joints[i].q;
	IF joints[i].bActive THEN	
///	
		// Set input based on velocity input u
//		qRef[i] := qRef[i] + fVelInput[i]*Ts;
//		qRef_t[i] := fVelInput[i];
//		qRef_tt[i] := (fVelInput[i]-fVelInputOld[i])/(Ts);
//		// Update old variable
//		fVelInputOld[i] := fVelInput[i];
		
///	
//-----------------------------------------------------------------------------------------------------------------------------------------		
			//traj
			//check if the pos input is changed
			IF bPositionModeExecute AND (NOT bExecuteReady[i]) THEN
				ft[i] := 0.0;
				fbTrajectoryGenerator[i].init(fqStartInit := joints[i].q + fDeflectionCompensation[i], fqFinalInit := fLimitedPosInput[i], ftFinalInit := ftf);
				bExecuteReady[i] := TRUE;
			END_IF
			IF bExecuteReady[i] THEN
				fbTrajectoryGenerator[i].getTrajectory(ftTraj := ft[i]);
				
//				qRef[i] := fbTrajectoryGenerator[i].fqPos;
//				qRef_t[i]:= fbTrajectoryGenerator[i].fqVel;
//				qRef_tt[i] :=  fbTrajectoryGenerator[i].fqAcc;
//-------------------------------------------------------------------------------------------------------------
				fPosDiff[i] := fbTrajectoryGenerator[i].fqPos - fDeflectionCompensation[i] - joints[i].q;
				qRef[i] := fbTrajectoryGenerator[i].fqPos - fDeflectionCompensation[i]; // joints[i].q + qRef_t[i]*Ts;	
				qRef_t[i] := KffPos[i]*fbTrajectoryGenerator[i].fqVel + KpPos[i]*fPosDiff[i] + KdPos[i]*(0.0 - q_t_Filtered[i]);
				qRef_tt[i] := fbTrajectoryGenerator[i].fqAcc;		
//------------------------------------------------------------------------------------------------------------------------------------	 
				ft[i] := ft[i]+Ts;
			ELSE
				qRef[i] := joints[i].q;
				qRef_t[i]:= 0.0;
				qRef_tt[i] :=  0.0;
				ft[i] := 0.0;
			END_IF
			
			IF (ft[i] > ftf) AND (ABS(fPosDiff[i]) < fPosThreshold) AND NOT bPositionModeExecute THEN //(ft[i] > ftf) remove
				bExecuteReady[i] := FALSE;
				ft[i] := 0.0;
			END_IF

//-----------------------------------------------------------------------------------------------------------------------------------------

////PD Control in position---------------------------------------------------------------------
		
//		qRef[i] := joints[i].q + qRef_t[i]*Ts;;
//		qRef_t[i] := KpPos[i]*(fPosInput[i] - joints[i].q) + KdPos[i]*(0.0 - q_t_Filtered[i]);
//		qRef_tt[i] :=  (qRef_t[i]-fVelInputOld[i])/(Ts);		
//		fVelInputOld[i] := qRef_t[i];

////--------------------------------------------------------------------------------------		
	ELSE
		bExecuteReady[i] := FALSE;
		fbTrajectoryGenerator[i].init(fqStartInit := joints[i].q, fqFinalInit := fLimitedPosInput[i], ftFinalInit := ftf);
		qRef[i] := joints[i].q;
		qRef_t[i]:= 0.0;
		qRef_tt[i] :=  0.0;	
	END_IF
	
END_FOR
END_METHOD

END_FUNCTION_BLOCK

// ---- POUs/FB_Joint.TcPOU
FUNCTION_BLOCK FB_Joint
VAR_INPUT
	bReset : BOOL;
	bEnable : BOOL;//e-stop can use this
	eRobotMode : E_RobotMode;


	bPositionModeExecute : BOOL;

	
	fGearRatio : LREAL := 1000.0;
	fTorqueScaling : LREAL := 1.0;
	
	qRef : LREAL;
	qRef_t : LREAL;
	qRef_tt : LREAL;
	fShaftAdditiveTorque : LREAL; // [Nm] on shaft
	fShaftAdditiveVelocity : LREAL; //deg/sec on shaft
	fShaftTorqueRef : LREAL; //Nm initialize with holding torque??
	
	fShaftAdditiveVelocityTest : LREAL; //deg/sec on shaft
	
	fTotalVelocityRef : LREAL;
	
	stJointParams : ST_JointParameters;
//	fOffset : LREAL;
	Ts : LREAL;
END_VAR
VAR_OUTPUT
	// eRobotMode : E_RobotMode;

	bActive : BOOL;
	bAxisStopped :BOOL;
	
	qRefLimited : LREAL;
	
	// Joint feedback
	q : LREAL;
	q_t : LREAL;
	tau : LREAL;
	fVelocityControllerShaftOutputTorque: LREAL; // [Nm] on shaft
END_VAR
VAR
	fAdditiveTorque : LREAL; // [Nm] on motor
	nAdditiveTorquePerc AT %Q* : INT;	
	
	nAdditiveVelocity AT %Q* : DINT; // rev/2^30 ms	
	
	nVelocityControllerOutputTorque AT %I*: INT;
 	fVelocityControllerOutputTorque: LREAL; // [Nm] on motor

	// Drive axis stuff
	axis : AXIS_REF;
	fbPower : MC_Power;
	fbReset : MC_Reset;
	
	//SoftStop
	fbStop : MC_Stop;	
	fDeceleration :LREAL := 100;
	fJerk :LREAL := 300;

	fOffset : LREAL;
	
	// External setpoint	
	fbExtSetPointGenEnable : MC_ExtSetPointGenEnable;
	fbExtSetPointGenDisable : MC_ExtSetPointGenDisable;
	fbReadParameterSet : MC_ReadParameterSet;
	stAxisParameterSet : ST_AxisParameterSet;
	bReadParameterSet : BOOL := TRUE;
	
	//move to position
	fbAxisMoveAbsolute : MC_MoveAbsolute;
	
	

	fbTorqueControl : FB_TorqueController;
	
	
//	//check move velocity command
//	fbMoveVelocity 	: MC_MoveVelocity;
//	fbSetOverride 	: MC_SetOverride;
//	bExecuteMoveVelocity : BOOL := FALSE;
//	bExecuteOverride : BOOL := FALSE;
//	fVelocityCmd : LREAL := 0.0;
//	stDirection : MC_Direction;
		
END_VAR

//IF NOT fbReadParameterSet.Busy AND NOT fbReadParameterSet.Error THEN
//	fbReadParameterSet(
//		Axis := axis,
//		Parameter := stAxisParameterSet,
//		Execute := TRUE
//	);
	
//ELSE
//	fbReadParameterSet(
//		Axis := axis,
//		Parameter := stAxisParameterSet,
//		Execute := FALSE
//	);
	
//END_IF


fbReadParameterSet(
	Axis := axis,
	Parameter := stAxisParameterSet,
	Execute := bReadParameterSet AND NOT fbReadParameterSet.Busy
);
IF NOT(fbReadParameterSet.Busy OR fbReadParameterSet.Error) THEN
	bReadParameterSet := FALSE;
END_IF

bAxisStopped := (
	axis.Status.NotMoving  
	AND NOT axis.Status.HasJob //this is necessary to avoid error while stopping when torque control mode is on
	AND ((eRobotMode = E_RobotMode.STOP) OR (eRobotMode = E_RobotMode.ESTOP))
	AND NOT(fbExtSetPointGenEnable.Enabled)
);

// Power and reset logic
fbPower(
	Axis := axis,
	Enable := (bEnable AND NOT bAxisStopped),
	Enable_Positive := (bEnable AND NOT bAxisStopped),
	Enable_Negative := (bEnable AND NOT bAxisStopped)
);

fbReset(
	Execute := bReset AND (bAxisStopped OR (eRobotMode = E_RobotMode.ESTOP)), //brest must also be set from fbrobot 
	Axis := axis
);

//you can't execute fbstop when fbExtSetPointGenEnable.Enabled ----> motion comands are not allowed for external setpoint generated axis
fbStop(
	Axis := axis,
	Execute := NOT(fbExtSetPointGenEnable.Enabled) AND (eRobotMode = E_RobotMode.STOP),
	Deceleration := fDeceleration,
	Jerk := fJerk
);

// Read power status
bActive := fbPower.Status;

//velocity control
// Enable external setpoint when on
fbExtSetPointGenDisable(
	Axis := axis,
	Execute := (eRobotMode <> E_RobotMode.VELOCITY) OR NOT(bActive)
);

fbExtSetPointGenEnable(
	Axis := axis,
	Execute := (eRobotMode = E_RobotMode.VELOCITY) AND bActive
);



qRefLimited := LIMIT(stJointParams.stPositionLimits.fMin, qRef, stJointParams.stPositionLimits.fMax);
fOffset := stJointParams.stOffsets.fCalibrationOffset + stJointParams.stOffsets.fPositionOffset;


IF bActive AND fbExtSetPointGenEnable.Enabled THEN		
	fShaftAdditiveVelocity := LIMIT(-stAxisParameterSet.fVeloMaximum, fShaftAdditiveVelocity, stAxisParameterSet.fVeloMaximum);
	
	nAdditiveVelocity := -TO_DINT(fShaftAdditiveVelocity*fGearRatio*CONSTANTS.VELOCITY_SCALING);
//	nAdditiveVelocity := -TO_DINT(fShaftAdditiveVelocityTest*fGearRatio*CONSTANTS.VELOCITY_SCALING);
	
	fTotalVelocityRef := -qRef_t - fShaftAdditiveVelocity; //this is only used for direction
//	fTotalVelocityRef := -qRef_t - fShaftAdditiveVelocityTest; //fShaftAdditiveVelocity;
	
	
	//Feed extrernal setpoints to axis interface
//	MC_ExtSetPointGenFeed(
//		Axis := axis,
//		Position := LIMIT(stAxisParameterSet.fEncSoftEndMin, fOffset - (qRef + fShaftAdditiveVelocity*Ts), stAxisParameterSet.fEncSoftEndMax),
//		Velocity := fTotalVelocityRef,
//		Acceleration := -qRef_tt,
//		Direction := getDirection(fTotalVelocityRef, -qRef_tt)
//	);

	
	MC_ExtSetPointGenFeed(
		Axis := axis,
		Position := fOffset - qRefLimited,
		Velocity := -qRef_t,
		Acceleration := -qRef_tt,
		Direction := getDirection(fTotalVelocityRef, -qRef_tt)
	);
	fAdditiveTorque := fShaftAdditiveTorque / fGearRatio;
	
	nAdditiveTorquePerc := TO_INT(
		RescaleRange(
			in := -fAdditiveTorque, //flip the direction
			in_min := -fTorqueScaling, 
			in_max := fTorqueScaling,
			out_min := -1000, 
			out_max := 1000 
		)
	);
		
	fVelocityControllerOutputTorque := 	RescaleRange(
		in := -TO_LREAL(nVelocityControllerOutputTorque), //flip the direction
		in_min := -1000, 
		in_max := 1000,
		out_min := -fTorqueScaling, 
		out_max := fTorqueScaling 
	);
	fVelocityControllerShaftOutputTorque :=fVelocityControllerOutputTorque*fGearRatio; 
ELSE
	nAdditiveTorquePerc := 0;
	fTotalVelocityRef := 0.0;
END_IF


//position control
fbAxisMoveAbsolute(
	Axis := axis,
	Execute := bPositionModeExecute AND (eRobotMode = E_RobotMode.POSITION) AND bActive,
	Position := (fOffset - qRefLimited), // (qRef - fOffset),
	Velocity := qRef_t,
	BufferMode := MC_BufferMode.MC_Aborting
);



////--------------------------------------------------------------------------------------------------------------------------
////check move velocity command
////position control
//IF fVelocityCmd <= 0.0 THEN
//	stDirection := MC_Direction.MC_Positive_Direction; //reverse due to our axis flip
//ELSE
//	stDirection := MC_Direction.MC_Negative_Direction; //reverse
//END_IF

//fbMoveVelocity(
//	Axis := axis,
//	Execute := bExecuteMoveVelocity AND (eRobotMode = E_RobotMode.POSITION) AND bActive,
//	Velocity := ABS(fVelocityCmd),
//	Direction := stDirection,
//	BufferMode := MC_BufferMode.MC_Aborting
//);
//fbSetOverride(Enable:= bExecuteOverride, Axis := axis);

////--------------------------------------------------------------------------------------------------------------------------


// Update axis data
axis();




//-----------------torque control
fbTorqueControl(
	Axis := axis,
	bEnable := bActive AND (eRobotMode = E_RobotMode.TORQUE),
	fShaftTorqueCmdNm := -fShaftTorqueRef, //negative sign is to change the direction
	fTorqueScaling := fTorqueScaling,
	fGearRatio := fGearRatio
);

// fbTorqueControl.readFeedback();







q := -axis.NcToPlc.ActPos + fOffset;
q_t := -axis.NcToPlc.ActVelo;
tau := - fbTorqueControl.fShaftTorqueFbkNm;

METHOD PRIVATE getDirection : DINT
VAR_INPUT
	fTargetVelocity : LREAL;
	fTargetAcceleration : LREAL;
END_VAR
IF fTargetVelocity = 0.0 AND fTargetAcceleration = 0.0 THEN
	// Standstill
	getDirection := 0;
	
ELSIF fTargetVelocity >= 0.0 THEN
	// Positive motion
	getDirection := 1;
	
ELSE
	// Negative motion
	getDirection := -1;
	
END_IF
END_METHOD

END_FUNCTION_BLOCK

// ---- POUs/FB_TorqueController.TcPOU
FUNCTION_BLOCK FB_TorqueController
VAR_INPUT
	bEnable: BOOL;
	fShaftTorqueCmdNm: LREAL; // Torque input in NM in the shaft after gearbox
	fTorqueScaling: LREAL:= 2.99;
	fVelocityLimitHigh: LREAL:= 100; // [mm/s]
	fVelocityLimitLow: LREAL:= 0; // [mm/s]
	fTorqueRamp: LREAL:= 100.0; // // [%/s] //10
	fGearRatio: LREAL := 1000;
	bStop: BOOL;
	bRelative: BOOL:= FALSE; //it should be false, but DS doesn't know why it was true by default
END_VAR
VAR_IN_OUT
	Axis: AXIS_REF;
END_VAR
VAR_OUTPUT
	fShaftSetTorqueNm: LREAL;
	fShaftTorqueFbkNm : LREAL;
	// Torque output
	bInTorque: BOOL;
	bBusy: BOOL;
	bActive: BOOL;
	bCommandAborted: BOOL;
	bError: BOOL;
	nErrId: UDINT;
	nMotorTempCelcius AT %I*: UINT;
	bDisabled : BOOL := TRUE;
END_VAR
VAR
	// Torque controller
	fbTorque: MC_TorqueControl;
	// Controller options
	stTorqueOptions: ST_TorqueControlOptions := (ManualTorqueStartValue:= 0, EnableManualTorqueStartValue:= FALSE); 	
	// Trigger on change in setpoint
	rTrigTorqueChange: R_Trig;
	
//	bEnable_last : BOOL := bEnable;
	fbEnableFalling : F_TRIG;
	fbReadDone 		: F_TRIG;
	fbWriteDone 	: F_TRIG;

	fTorqueCmdNm: LREAL; // Torque input in NM
	fTorqueFbkNm: LREAL; // Torque output
	
	// Setpoint
	fSetTorquePerc : LREAL;
	fSetTorqueNm: LREAL;
	
	fTorqueCmdPercent: LREAL; // [%] Torque
	fTorqueCmdPercentOld: LREAL; // [%] Torque
	
	// Torque feedback
	fTorqueFbkPerc AT %I*: INT;	
	// Torque feedback
	nFastStopState AT %I*: UINT;
	nAccFbk AT %I*: DINT;	
	nVelFbk AT %I*: DINT;
	

	fTorqueFbkNmFiltered : LREAL;
	
	// Stop handling
	mcStop : MC_Stop;
	bStopDone           : BOOL;
	bStopBusy           : BOOL;
	bStopActive         : BOOL;
	bStopCommandAborted : BOOL;
	bStopError          : BOOL;
	nStopErrorID        : UDINT;
	rTrigStop: R_TRIG;
	fbMcPower : MC_POWER;
	
	eState: UDINT;
	
	
	//read  and write drive operation mode
	fbMC_ReadDriveOperationMode : MC_ReadDriveOperationMode;
	fbMC_WriteDriveOperationMode : MC_WriteDriveOperationMode;
//	bReadDriveOperationMode : BOOL := FALSE;
//	bWriteDriveOperationMode : BOOL := FALSE;

	
END_VAR

// Read torque feedback
 readFeedback();
 
fTorqueCmdNm := fShaftTorqueCmdNm/fGearRatio;



// Scale torque command in NM to percentage
fTorqueCmdPercent:= RescaleRange(fTorqueCmdNm, -fTorqueScaling, fTorqueScaling, -100, 100);
// Set falling edge before new setpoint
IF(fTorqueCmdPercent <> fTorqueCmdPercentOld) AND bEnable THEN
	
	fbTorque(Axis:= Axis, Execute:= FALSE);
	
END_IF
// Store current torque as old torque
fTorqueCmdPercentOld:= fTorqueCmdPercent;	


// Torque testing
fbTorque(
	Axis:= Axis,
	Execute:= bEnable,
	Relative:= bRelative, // Torque setpoint relative to current torque load???
	Torque:= fTorqueCmdPercent,
	TorqueRamp:= fTorqueRamp,
	VelocityLimitHigh:= fVelocityLimitHigh,
	VelocityLimitLow:= fVelocityLimitLow,
	BufferMode:= MC_BufferMode.MC_Aborting, // Abort current if new cmd
	Options:= stTorqueOptions,
	InTorque => bInTorque,
	Busy => bBusy,
	Active => bActive,
	CommandAborted => bCommandAborted,
	Error => bError,
	ErrorId => nErrId
);



// Torque setpoints (% and NM)
fSetTorquePerc:= Axis.NcToPlc.SetTorque;
fSetTorqueNm:= RescaleRange(fSetTorquePerc, -100, 100, -fTorqueScaling, fTorqueScaling);
fShaftSetTorqueNm := fSetTorqueNm*fGearRatio;



//IF bEnable THEN
//	bReadDriveOperationMode := FALSE;
//	bWriteDriveOperationMode := FALSE;
//ELSE 
//	bReadDriveOperationMode := TRUE;//to see if the drive operation mode is in velocity control mode
//	bWriteDriveOperationMode := TRUE;	//to bring it to velocity control if the drive operation mode is not in velocity control mode
//END_IF

IF bEnable THEN
	bDisabled := FALSE;
END_IF

fbEnableFalling(CLK := bEnable);
IF fbEnableFalling.Q OR fbWriteDone.Q THEN
//	bReadDriveOperationMode := TRUE; // to see if the drive operation mode is in velocity control mode
	fbMC_ReadDriveOperationMode.Execute := TRUE;
END_IF

fbMC_ReadDriveOperationMode(
		Axis := axis
//		Execute := bReadDriveOperationMode
);
//bReadDriveOperationMode := FALSE; // to see if the drive operation mode is in velocity control mode	
fbMC_ReadDriveOperationMode.Execute := FALSE;

fbReadDone(CLK := fbMC_ReadDriveOperationMode.Busy);
IF fbReadDone.Q AND NOT(bEnable) THEN
	IF (fbMC_ReadDriveOperationMode.DriveOperationMode = E_DriveOperationMode.DriveOperationMode_Velo1) THEN
		bDisabled := TRUE;
	ELSE
		fbMC_WriteDriveOperationMode.Execute := TRUE;
//		bWriteDriveOperationMode := TRUE;
	END_IF
END_IF

//IF (fbMC_ReadDriveOperationMode.Busy OR fbMC_ReadDriveOperationMode.Error) THEN 
//	bReadDriveOperationMode := FALSE;//attempt once again
//END_IF

//IF THEN
//END_IF
fbMC_WriteDriveOperationMode(
	Axis := axis,
	DriveOperationMode := E_DriveOperationMode.DriveOperationMode_Velo1
);
fbMC_WriteDriveOperationMode.Execute := FALSE;

fbWriteDone(CLK := fbMC_WriteDriveOperationMode.Busy);

//IF (fbMC_WriteDriveOperationMode.Busy OR fbMC_WriteDriveOperationMode.Error) THEN
//	bWriteDriveOperationMode := FALSE;//attempt once again
//END_IF

METHOD readFeedback : BOOL
VAR_INPUT

END_VAR
// S-0-0084 Torque feedback value
// The parameter contains the current in one-tenth of a percent relative to P-0-0094 (Configured channel peak torque)
// (Hence signal range [-1000, 1000])
fTorqueFbkNm := RescaleRange(INT_TO_LREAL(fTorqueFbkPerc), -1000, 1000, -fTorqueScaling, fTorqueScaling);



// Calculate shaft torque after gearbox
fTorqueFbkNmFiltered := fTorqueFbkNm;
fShaftTorqueFbkNm:= fTorqueFbkNmFiltered * fGearRatio;
END_METHOD

END_FUNCTION_BLOCK

// ---- POUs/RescaleRange.TcPOU
FUNCTION RescaleRange : LREAL
VAR_INPUT
	in: LREAL;
	in_min: LREAL;
	in_max: LREAL;
	out_min: LREAL;
	out_max: LREAL;
END_VAR

in := LIMIT(in_min, in, in_max);
RescaleRange := LIMIT(out_min, (out_min + (in - in_min)*(out_max-out_min)/(in_max-in_min)), out_max);

END_FUNCTION

// ---- POUs/FB_LowPassFilter.TcPOU
FUNCTION_BLOCK FB_LowPassFilter
VAR_INPUT
END_VAR
VAR_OUTPUT
	bInitialized 	: BOOL := FALSE;
	bInitError		: BOOL := FALSE;
	fOut 			: LREAL := 0.0;
END_VAR
VAR
	a : LREAL := 1.0;
	b : LREAL := 0.0;
	c : LREAL := 0.0;
	
	fOut_t2 : LREAL := 0.0;
END_VAR

METHOD PUBLIC init : BOOL
VAR_INPUT
	stParams : REFERENCE TO ST_FilterParams;
END_VAR
VAR

END_VAR
bInitError := FALSE;

CASE stParams.eOrder OF
E_FilterOrder.eFirst:
	initFirstOrder(stParams);

E_FilterOrder.eSecond:
	initSecondOrder(stParams);
	
ELSE	
	bInitError := TRUE;
	init := bInitialized := FALSE;
	a := 1.0;
	b := 0.0;
	c := 0.0;
	RETURN;
END_CASE


IF bInitError OR (a <= 0.0) OR (a > 1.0) THEN
	bInitError := TRUE;
	init := bInitialized := FALSE;
	a := 1.0;
	b := 0.0;
	c := 0.0;
	RETURN;
END_IF

fOut := stParams.fInitialValue;
init := bInitialized := TRUE;
END_METHOD

METHOD PRIVATE initFirstOrder
VAR_INPUT
	stParams : REFERENCE TO ST_FilterParams;
END_VAR
VAR
	wc 		: LREAL;

	tmp1 	: LREAL;
	tmp2	: LREAL;
END_VAR
wc := stParams.fCutoff*2.0*PI;

tmp1 := wc*stParams.fDeltaTime;

tmp2 := 1 + tmp1;

IF (tmp2 <= 0.0) THEN
	bInitError := TRUE;
	bInitialized := FALSE;
	a := 1.0;
	b := 0.0;
	c := 0.0;
	RETURN;
END_IF

a := tmp1/tmp2;
b := 1.0 - a;
c := 0.0;
END_METHOD

METHOD PRIVATE initSecondOrder
VAR_INPUT
	stParams : REFERENCE TO ST_FilterParams;
END_VAR
VAR
	wc 		: LREAL;

	tmp1 	: LREAL;
	tmp2 	: LREAL;
	tmp3	: LREAL;
END_VAR
wc := stParams.fCutoff*2.0*PI;

tmp1 := wc*stParams.fDeltaTime;
tmp2 := EXPT(tmp1, 2.0);
tmp3 := 1.0 + 2.0*wc*stParams.fDeltaTime*stParams.fDampingRatio + tmp2;

IF (tmp3 <= 0.0) THEN
	bInitError := TRUE;
	bInitialized := FALSE;
	a := 1.0;
	b := 0.0;
	c := 0.0;
	RETURN;
END_IF

a := tmp2/tmp3;
b := 2.0*(1.0 + tmp1)/tmp3;
c := 1.0 - a - b;
END_METHOD

METHOD PUBLIC update : LREAL
VAR_INPUT
	fIn : LREAL;
END_VAR
VAR
	tmp : LREAL;
END_VAR

tmp := fOut;

update := fOut := a*fIn + b*fOut + c*fOut_t2;

fOut_t2 := tmp;
END_METHOD

END_FUNCTION_BLOCK

// ---- POUs/FB_TrajectoryGenerator.TcPOU
FUNCTION_BLOCK FB_TrajectoryGenerator
VAR_INPUT
END_VAR
VAR_OUTPUT
	fqPos : LREAL; //joint pos
	fqVel : LREAL; //joint vel
	fqAcc : LREAL; //joint acc
END_VAR
VAR
	fqStart : LREAL; //start pos
	fqFinal : LREAL; //goal ¨pos
	ftFinal : LREAL; //final time	
	

	a0  : LREAL := 0.0;
	a1  : LREAL := 0.0;
	a2  : LREAL := 0.0;
	a3  : LREAL := 0.0;
	a4  : LREAL := 0.0;
	a5  : LREAL := 0.0;
	
	
END_VAR

METHOD getTrajectory : BOOL
VAR_INPUT
	ftTraj : LREAL; // traj point
END_VAR

IF ftTraj <= ftFinal THEN
	fqPos := a0 + a1*EXPT(ftTraj,1) +  a2*EXPT(ftTraj,2) + a3*EXPT(ftTraj,3) + a4*EXPT(ftTraj,4) + a5*EXPT(ftTraj,5);
	fqVel := a1 +  2*a2*EXPT(ftTraj,1) + 3*a3*EXPT(ftTraj,2) + 4*a4*EXPT(ftTraj,3) + 5*a5*EXPT(ftTraj,4);
	fqAcc := 2*a2 + 2*3*a3*EXPT(ftTraj,1) + 3*4*a4*EXPT(ftTraj,2) + 4*5*a5*EXPT(ftTraj,3);
ELSE
	fqPos := fqFinal;
	fqVel := 0.0;
	fqAcc := 0.0;
END_IF
END_METHOD

METHOD init : BOOL
VAR_INPUT
	fqStartInit : LREAL; //start pos
	fqFinalInit : LREAL; //goal ¨pos
	ftFinalInit : LREAL; //final time	
END_VAR

fqStart := fqStartInit;
fqFinal := fqFinalInit;
ftFinal := ftFinalInit;

a0 := fqStartInit;
a1 := 0.0;
a2 := 0.0;
a3 := (10*(fqFinalInit - fqStartInit))/EXPT(ftFinalInit,3);
a4 := -(15*(fqFinalInit - fqStartInit))/EXPT(ftFinalInit,4);
a5 :=  (6*(fqFinalInit - fqStartInit))/EXPT(ftFinalInit,5);
END_METHOD

END_FUNCTION_BLOCK

// ---- MATRIX/FB_Vector3.TcPOU
FUNCTION_BLOCK PUBLIC FB_Vector3 EXTENDS ExternalStaticMatrix
VAR_INPUT
END_VAR
VAR_OUTPUT
END_VAR
VAR
	data_array : ARRAY [0..2] OF LREAL;
END_VAR

METHOD FB_init : BOOL
VAR_INPUT
	bInitRetains : BOOL; // if TRUE, the retain variables are initialized (warm start / cold start)
	bInCopyCode : BOOL;  // if TRUE, the instance afterwards gets moved into the copy code (online change)
END_VAR
VAR
END_VAR
Init(ADR(data_array), 3, 1);
Clear();
END_METHOD

PROPERTY PUBLIC X : LREAL
GET
X := GetI(0);
END_GET
SET
SetI(0, X);
END_SET
END_PROPERTY

PROPERTY PUBLIC Y : LREAL
GET
Y := GetI(1);
END_GET
SET
SetI(1, Y);
END_SET
END_PROPERTY

PROPERTY PUBLIC Z : LREAL
GET
Z := GetI(2);
END_GET
SET
SetI(2, Z);
END_SET
END_PROPERTY

END_FUNCTION_BLOCK

// ---- POUs/P_HMI.TcPOU
PROGRAM P_HMI
VAR
	i : UINT;
	fbSafety_GroupPort_ErrAck 		: TOF := (PT := T#0.5S);
	fbSafety_EStopRestart 			: TOF := (PT := T#0.5S);
	fbSafety_Drive_Axis_ErrReset 	: TOF := (PT := T#0.5S);
END_VAR

//------------------------------------------------------
//--------------------- HMI to PLC ---------------------

IF HmiToPlc.bPositionMode THEN
	// Attempt to enable position mode
	MAIN.robot.eRobotModeCmd := E_RobotMode.POSITION;
END_IF
HmiToPlc.bPositionMode := FALSE;

IF HmiToPlc.bVelocityMode THEN
	// Attempt to enable velocity mode
	MAIN.robot.eRobotModeCmd := E_RobotMode.VELOCITY;
END_IF
HmiToPlc.bVelocityMode := FALSE;

IF HmiToPlc.bTorqueMode THEN
	// Attempt to enable torque mode
//	MAIN.robot.eRobotModeCmd := E_RobotMode.TORQUE;	
END_IF
HmiToPlc.bTorqueMode := FALSE;

IF HmiToPlc.bSoftStop THEN
	// Stop
	MAIN.robot.eRobotModeCmd := E_RobotMode.STOP;	
END_IF
HmiToPlc.bSoftStop := FALSE;

MAIN.robot.bReset := HmiToPlc.bReset;
HmiToPlc.bReset := FALSE;

IF HmiToPlc.bEnable THEN
	// Enable joints
	MAIN.robot.bEnable := TRUE;
END_IF
HmiToPlc.bEnable := FALSE;

MAIN.robot.bPositionModeExecute := HmiToPlc.bPositionModeExecute;
HmiToPlc.bPositionModeExecute := FALSE;

fbSafety_GroupPort_ErrAck(IN := HmiToPlc.bSafety_GroupPort_ErrAck);
Safety.TS_Q_Safety_GroupPort_ErrAck := fbSafety_GroupPort_ErrAck.Q;
HmiToPlc.bSafety_GroupPort_ErrAck := FALSE;

fbSafety_EStopRestart(IN := HmiToPlc.bSafety_EStopRestart);
Safety.TS_Q_Safety_EStopRestart := fbSafety_EStopRestart.Q;
HmiToPlc.bSafety_EStopRestart := FALSE;

fbSafety_Drive_Axis_ErrReset(IN := HmiToPlc.bSafety_Drive_Axis_ErrReset);
Safety.TS_Q_Safety_Drive_Axis_ErrReset := fbSafety_Drive_Axis_ErrReset.Q;
HmiToPlc.bSafety_Drive_Axis_ErrReset := FALSE;

FOR i := 0 TO 2 DO
	MAIN.fPosInput[i] := HmiToPlc.fPosInput[i];
	MAIN.fVelInput[i] := HmiToPlc.fVelInput[i];
END_FOR

//------------------------------------------------------
//--------------------- PLC to HMI ---------------------

PlcToHmi.bPositionMode := (MAIN.robot.eRobotMode = E_RobotMode.POSITION);
PlcToHmi.bVelocityMode := (MAIN.robot.eRobotMode = E_RobotMode.VELOCITY);
PlcToHmi.bTorqueMode := (MAIN.robot.eRobotMode = E_RobotMode.TORQUE);

FOR i := 0 TO 2 DO
	PlcToHmi.fPosFb[i] := MAIN.robot.q[i];
	PlcToHmi.fVelFb[i] := MAIN.robot.q_t[i];
	PlcToHmi.fTauFb[i] := MAIN.robot.tau[i];
END_FOR

PlcToHmi.bAnyJointActive := MAIN.robot.bAnyJointActive;
PlcToHmi.bSafety_EStopError := Safety.TS_I_Safety_EStopError;
PlcToHmi.bSafety_EStopOK := Safety.TS_I_Safety_EStopOK;

END_PROGRAM

// ---- MATRIX/AccelerometerReadings.TcPOU
FUNCTION AccelerometerReadings : BOOL
VAR_INPUT
	q : ARRAY [0..2] OF LREAL;
	qdot : ARRAY [0..2] OF LREAL;
	qddot : ARRAY [0..2] OF LREAL;
	L : ARRAY [0..2] OF LREAL;
	Tip_to_IMU : REFERENCE TO ARRAY [0..2] OF FB_Vector3;
	AccelerometerReadingsOut : REFERENCE TO ARRAY [0..2] OF FB_Vector3;
	gravity_vector : REFERENCE TO FB_Vector3;
	
END_VAR
VAR
	
	z0 : FB_Vector3 := (X := 0, Y := 0, Z := 1);
	
	T_from_i_1_to_i : FB_Matrix4x4;
	Rot : FB_Matrix3x3;
	Rot_Trans : TransposeMatrixAccessor;
	Rot_IMU_Joint : FB_Matrix3x3;
	w : ARRAY [0..2] OF FB_Vector3;
	wdot : ARRAY [0..2] OF FB_Vector3;
	vdot : ARRAY [0..2] OF FB_Vector3;
	vIMUdot : ARRAY [0..2] OF FB_Vector3;	

	p : FB_Vector3; 

	i : USINT;
	
	
	prod_z0_qdot : FB_Vector3;	
	

	tmp : SubMatrixAccessor;
	
	prod_z0_qddot : FB_Vector3;	

		
		
	prod_Rottrans_grav : FB_Vector3;
	cross_wdot_p : FB_Vector3;
	cross_w_p : FB_Vector3;
	cross_w_w_p : FB_Vector3;
	
	cross_wdot_imu : FB_Vector3;
	cross_w_imu : FB_Vector3;
	cross_w_w_imu : FB_Vector3;

	sum_w_prod_z0_qdot : FB_Vector3;
	
	sum_wdot_prod_z0_qddot_cross_w_prod_z0_qdot : FB_Vector3;
	cross_w_prod_z0_qdot : FB_Vector3;
	
	prod_Rottrans_vdot : FB_Vector3;

	
	
	
END_VAR


//gravity_vector.SetI(0, 0);
//gravity_vector.SetI(1, 9.8*1);
//gravity_vector.SetI(2, 0);


//z0.SetI(0,0);
//z0.SetI(1,0);
//z0.SetI(2,1);

Rot_IMU_Joint.SetRC(0,0,0);
Rot_IMU_Joint.SetRC(0,1,0);
Rot_IMU_Joint.SetRC(0,2,1);
Rot_IMU_Joint.SetRC(1,0,1);
Rot_IMU_Joint.SetRC(1,1,0);
Rot_IMU_Joint.SetRC(1,2,0);
Rot_IMU_Joint.SetRC(2,0,0);
Rot_IMU_Joint.SetRC(2,1,1);
Rot_IMU_Joint.SetRC(2,2,0);

FOR i:=0 TO 2 DO
	
   	F_DH(theta:= q[i],d:=0,a:=L[i],alpha:=0,T_from_i_1_to_i);
	tmp := T_from_i_1_to_i.GetSubMatrixAccessor(RowStart:=0,RowCount:=3,ColStart:=0,ColCount:=3);
	tmp.CopyTo(Rot);
	Rot_Trans := Rot.GetTransposeMatrixAccessor();
	
	p.SetI(0,L[i]);
	p.SetI(1,0);
	p.SetI(2,0);
	
	IF i > 0 THEN
//        w(:, i) =  R'*(w(:, i-1) + z0.*qdot(i));
		z0.CopyTo(prod_z0_qdot); 								// z0.*qdot(i)
		prod_z0_qdot.Scale(qdot[i]);
		prod_z0_qdot.CopyTo(sum_w_prod_z0_qdot);
		sum_w_prod_z0_qdot.ElementSum(w[i-1]);
		Matrix_Product(Rot_Trans,sum_w_prod_z0_qdot,w[i]); 



//        wdot(:, i) = R'*(wdot(:, i-1) +  z0.*qddot(i) + ...
//            cross(w(:, i-1), z0.*qdot(i)));
		z0.CopyTo(prod_z0_qddot); 								
		prod_z0_qddot.Scale(qddot[i]);		
		F_Cross2(w[i-1],prod_z0_qdot,cross_w_prod_z0_qdot);		
		
		wdot[i-1].CopyTo(sum_wdot_prod_z0_qddot_cross_w_prod_z0_qdot);
		sum_wdot_prod_z0_qddot_cross_w_prod_z0_qdot.ElementSum(prod_z0_qddot);
		sum_wdot_prod_z0_qddot_cross_w_prod_z0_qdot.ElementSum(cross_w_prod_z0_qdot);
		Matrix_Product(Rot_Trans,sum_wdot_prod_z0_qddot_cross_w_prod_z0_qdot,wdot[i]); 

//        vdot(:,i) = R'*vdot(:,i-1) + cross(wdot(:,i), p) + ...
//            cross(w(:,i), cross(w(:,i),p));-----------------------------------------------------------------
			
		Matrix_Product(Rot_Trans,vdot[i-1],prod_Rottrans_vdot); 				
		F_Cross2(wdot[i],p,cross_wdot_p);
		F_Cross2(w[i],p,cross_w_p);
		F_Cross2(w[i],cross_w_p,cross_w_w_p);
		
		prod_Rottrans_vdot.CopyTo(vdot[i]);
		vdot[i].ElementSum(cross_wdot_p);
		vdot[i].ElementSum(cross_w_w_p);
		
		

		
		


//        vIMUdot(:,i) = vdot(:,i) + cross(wdot(:,i),Tip_to_IMU(:,i)) + ...
//            cross(w(:,i),cross(w(:,i),Tip_to_IMU(:,i)));

		F_Cross2(wdot[i],Tip_to_IMU[i],cross_wdot_imu);
		F_Cross2(w[i],Tip_to_IMU[i],cross_w_imu);
		F_Cross2(w[i],cross_w_p,cross_w_w_imu);
		
		
		vdot[i].CopyTo(vIMUdot[i]);
		vIMUdot[i].ElementSum(cross_wdot_imu);
		vIMUdot[i].ElementSum(cross_w_w_imu);





	ELSE		
//		        w(:, i) =  R'*(z0.*qdot(i));
		z0.CopyTo(prod_z0_qdot); 								// z0.*qdot(i)
		prod_z0_qdot.Scale(qdot[i]);
		Matrix_Product(Rot_Trans,prod_z0_qdot,w[i]); // R'*(z0.*qdot(i));

//        wdot(:, i) = R'*(z0.*qddot(i));
		z0.CopyTo(prod_z0_qddot); 								
		prod_z0_qddot.Scale(qddot[i]);									
		Matrix_Product(Rot_Trans,prod_z0_qddot,wdot[i]); // R'*(z0.*qddot(i));	


//        vdot(:,i) = R'*grav + cross(wdot(:,i), p) + ...
//            cross(w(:,i), cross(w(:,i),p));
		Matrix_Product(Rot_Trans,gravity_vector,prod_Rottrans_grav);
		F_Cross2(wdot[i],p,cross_wdot_p);
		F_Cross2(w[i],p,cross_w_p);
		F_Cross2(w[i],cross_w_p,cross_w_w_p);
		
		
		prod_Rottrans_grav.CopyTo(vdot[i]);
		vdot[i].ElementSum(cross_wdot_p);
		vdot[i].ElementSum(cross_w_w_p);


//        vIMUdot(:,i) = vdot(:,i) + cross(wdot(:,i),Tip_to_IMU(:,i)) + ...
//            cross(w(:,i),cross(w(:,i),Tip_to_IMU(:,i)));

		F_Cross2(wdot[i],Tip_to_IMU[i],cross_wdot_imu);
		F_Cross2(w[i],Tip_to_IMU[i],cross_w_imu);
		F_Cross2(w[i],cross_w_p,cross_w_w_imu);
		
		
		vdot[i].CopyTo(vIMUdot[i]);
		vIMUdot[i].ElementSum(cross_wdot_imu);
		vIMUdot[i].ElementSum(cross_w_w_imu);



	END_IF	
	Matrix_Product(Rot_IMU_Joint,vIMUdot[i],AccelerometerReadingsOut[i]);	
	
END_FOR;

END_FUNCTION

// ---- MATRIX/FB_Matrix4x4.TcPOU
FUNCTION_BLOCK PUBLIC FB_Matrix4x4 EXTENDS ExternalStaticMatrix
VAR_INPUT
END_VAR
VAR_OUTPUT
END_VAR
VAR
	data_array : ARRAY [0..15] OF LREAL;
END_VAR

METHOD FB_init : BOOL
VAR_INPUT
	bInitRetains : BOOL; // if TRUE, the retain variables are initialized (warm start / cold start)
	bInCopyCode : BOOL;  // if TRUE, the instance afterwards gets moved into the copy code (online change)
END_VAR
VAR
END_VAR
Init(ADR(data_array), 4, 4);
Clear();
END_METHOD

END_FUNCTION_BLOCK

// ---- MATRIX/FB_Matrix3x3.TcPOU
FUNCTION_BLOCK PUBLIC FB_Matrix3x3 EXTENDS ExternalStaticMatrix
VAR_INPUT
END_VAR
VAR_OUTPUT
END_VAR
VAR
	data_array : ARRAY [0..8] OF LREAL;
END_VAR

METHOD FB_init : BOOL
VAR_INPUT
	bInitRetains : BOOL; // if TRUE, the retain variables are initialized (warm start / cold start)
	bInCopyCode : BOOL;  // if TRUE, the instance afterwards gets moved into the copy code (online change)
END_VAR
VAR
END_VAR
Init(ADR(data_array), 3, 3);
Clear();
END_METHOD

END_FUNCTION_BLOCK

// ---- MATRIX/F_DH.TcPOU
FUNCTION F_DH : BOOL
VAR_INPUT
	theta : LREAL;
	d : LREAL;
	a : LREAL;
	alpha : LREAL;
	F_DH_OUT : REFERENCE TO FB_Matrix4x4;
END_VAR
VAR
END_VAR


F_DH_OUT.SetRC(0, 0, COS(theta));
F_DH_OUT.SetRC(0, 1, -SIN(theta)*COS(alpha));
F_DH_OUT.SetRC(0, 2, SIN(theta)*SIN(alpha));
F_DH_OUT.SetRC(0, 3, a*COS(theta));

F_DH_OUT.SetRC(1, 0, SIN(theta));
F_DH_OUT.SetRC(1, 1, COS(theta)*COS(alpha));
F_DH_OUT.SetRC(1, 2, -COS(theta)*SIN(alpha));
F_DH_OUT.SetRC(1, 3, a*SIN(theta));


F_DH_OUT.SetRC(2, 0, 0);
F_DH_OUT.SetRC(2, 1, SIN(alpha));
F_DH_OUT.SetRC(2, 2, COS(alpha));
F_DH_OUT.SetRC(2, 3, d);

F_DH_OUT.SetRC(3, 0, 0);
F_DH_OUT.SetRC(3, 1, 0);
F_DH_OUT.SetRC(3, 2, 0);
F_DH_OUT.SetRC(3, 3, 1);

END_FUNCTION

// ---- MATRIX/F_Cross2.TcPOU
FUNCTION F_Cross2 : BOOL
VAR_INPUT
	vecA 	: REFERENCE TO FB_Vector3;
	vecB 	: REFERENCE TO FB_Vector3;
	res 	: REFERENCE TO FB_Vector3;
END_VAR
VAR
	cross_AB : ARRAY[0..1] OF POINTER TO Matrix := [ADR(vecA), ADR(vecB)];
END_VAR

Vector_CrossProduct(res, cross_AB);

END_FUNCTION

// ---- IMU/POUs/BackgroundCOM.TcPOU
PROGRAM BackgroundCOM
VAR
	i : DINT;
	

END_VAR

FOR i := 0 TO 2 DO
	IMU.fbStim300[i](fJointAccAtImuX := MAIN.fGainAccXYZ[0]*MAIN.AccelerometerReadingsOutWithoutGravity[i].X/CONSTANTS.GRAVITY,//represent in terms of Gravuty constant
					fJointAccAtImuY := MAIN.fGainAccXYZ[1]*MAIN.AccelerometerReadingsOutWithoutGravity[i].Y/CONSTANTS.GRAVITY,
					fJointAccAtImuZ := MAIN.fGainAccXYZ[2]*MAIN.AccelerometerReadingsOutWithoutGravity[i].Z/CONSTANTS.GRAVITY);
END_FOR

END_PROGRAM

// ---- IMU/POUs/FB_MapStim300.TcPOU
FUNCTION_BLOCK FB_MapStim300
VAR_INPUT
	stFilterParams : ST_FilterParams;
	
	fbFilter : FB_LowPassFilter;
	
	fJointAccAtImuX : LREAL := 0.0;//in terms of g
	fJointAccAtImuY : LREAL := 0.0;//in terms of g
	fJointAccAtImuZ : LREAL := 0.0;//in terms of g
	
	
END_VAR
VAR_OUTPUT
	ImuData : ST_IMUData;
	
	fRollDegFiltered : LREAL;
	fRollDeg : LREAL;
	fPitchDeg : LREAL;
END_VAR

VAR
		

	//serial communication with el6022
	fbGetSerialData : FB_GetSerialData;	
	ImuRawDataFrame : tDataFrame;
	
	fbEL6022Ctrl       : SerialLineControl;
	bEL6022CtrlError   : BOOL;
   	eEL6022CtrlErrorID : ComError_t;
   
	(* I/O variables for a EL6022 terminal*)
	stIn_EL6022 AT %I*    : EL6inData22B; 		(* linked to the EL6022 in the TwinCAT System Manager *)
	stOut_EL6022 AT %Q*    : EL6outData22B;		(* linked to the EL6022 in the TwinCAT System Manager *)
	
	RxBufferEL : ComBuffer; (* Receive data buffer; used with all receive function blocks *)
	TxBufferEL : ComBuffer; (* Transmit data buffer; used with all receive function blocks *)

	

	fbTimer : TON := (PT := T#1S);
	nCounter : DINT;
	fSampleRate : LREAL;
	
	//COmplementary filter
	fbAccelerometer : FB_AccelerometerAngle;
	fbComplementaryFilterRoll : FB_ComplementaryFilter := (fFilterRatio:=0.98);
	fbComplementaryFilterPitch : FB_ComplementaryFilter := (fFilterRatio:=0.98);
	
	// Task cycle time monitoring
	bFirstRun 		: BOOL := TRUE;
	bFirstSample 	: BOOL := TRUE;
	Ts : LREAL := 0.01;
	fbGetCurrentTaskIdx : GETCURTASKINDEX;
	bCycleTimeExceeded : BOOL;
	nCycleCount : UDINT;
	
END_VAR

VAR CONSTANT
	header : BYTE := 16#AF;
	nDataSize : UDINT := SIZEOF(tDataFrame);
	fRatioGyro : LREAL := 1.0/EXPT(2,14);
	fRatioAcc : LREAL := 1.0/EXPT(2,19);
END_VAR

IF bFirstRun THEN
	getSampleTIme();
	bFirstRun:= FALSE;
END_IF

fbEL6022Ctrl(
   Mode:= SERIALLINEMODE_EL6_22B, 
   pComIn:= ADR(stIn_EL6022), 
   pComOut:= ADR(stOut_EL6022), 
   SizeComIn:= SIZEOF(stIn_EL6022), 
   Error=> bEL6022CtrlError, 
   ErrorID=> eEL6022CtrlErrorID, 
   TxBuffer:= TxBufferEL, 
   RxBuffer:= RxBufferEL
);

nCounter := nCounter + 1;
fbTimer(IN := TRUE);
IF fbTimer.Q THEN
	fbTimer(IN := FALSE);
	fSampleRate := 1.0/TO_LREAL(nCounter);
	nCounter := 0;
END_IF

fbGetSerialData(
	pHeader := ADR(header),
	cbHeaderSize := 1,
	cbPacketSize := nDataSize,
	stRxBuffer := RxBufferEL,
	pDataBuffer := ADR(ImuRawDataFrame),
	cbDataBufferSize := nDataSize
);

IF fbGetSerialData.NewData THEN
	mapStim300(
		in := ADR(ImuRawDataFrame),
		out := ImuData
	);
	
	fbAccelerometer(fAx:=ImuData.stAcc.x - fJointAccAtImuX,fAy:=ImuData.stAcc.y - fJointAccAtImuY,fAz:=ImuData.stAcc.z - fJointAccAtImuZ); //subtract joint induced acc in all axis
	
	IF bFirstSample THEN
		bFirstSample := FALSE;
		stFilterParams.fCutoff := 10;//Hz
		stFilterParams.fDeltaTime := Ts;
		stFilterParams.fInitialValue := fRollDeg;
		fbFilter.init(stParams:=stFilterParams);
	END_IF
END_IF

fbComplementaryFilterRoll(fAccAngle:=fbAccelerometer.fRoll,fGyroRate:=ImuData.stGyro.x*CONSTANTS.DEG_TO_RAD,fStepTime:=Ts,fAngle=>ImuData.fRoll);
fbComplementaryFilterPitch(fAccAngle:=fbAccelerometer.fPitch,fGyroRate:=ImuData.stGyro.y*CONSTANTS.DEG_TO_RAD,fStepTime:=Ts,fAngle=>ImuData.fPitch);

fRollDeg := ImuData.fRoll * CONSTANTS.RAD_TO_DEG;

//Low pass filter
fRollDegFiltered := fbFilter.update(fRollDeg);




fPitchDeg := ImuData.fPitch * CONSTANTS.RAD_TO_DEG;

ACTION getSampleTIme:
// Get sample time of current task
fbGetCurrentTaskIdx();
bCycleTimeExceeded := _TaskInfo[fbGetCurrentTaskIdx.index].CycleTimeExceeded;
nCycleCount := _TaskInfo[fbGetCurrentTaskIdx.index].CycleCount;
Ts := UDINT_TO_LREAL(_TaskInfo[fbGetCurrentTaskIdx.index].CycleTime/10)/1E6;
//stFilterParams.fSamplingRate := Ts;
END_ACTION

METHOD PUBLIC mapStim300
VAR_INPUT
	in 	: POINTER TO BYTE;
	out : REFERENCE TO ST_ImuData;
END_VAR
	
	out.stGyro.x := TO_LREAL(F_Merge24BitSigned(in[1], in[2], in[3]))*fRatioGyro;
	out.stGyro.y := TO_LREAL(F_Merge24BitSigned(in[4], in[5], in[6]))*fRatioGyro;
	out.stGyro.z := TO_LREAL(F_Merge24BitSigned(in[7], in[8], in[9]))*fRatioGyro;
	
	out.stAcc.x := TO_LREAL(F_Merge24BitSigned(in[11], in[12], in[13]))*fRatioAcc;
	out.stAcc.y := TO_LREAL(F_Merge24BitSigned(in[14], in[15], in[16]))*fRatioAcc;
	out.stAcc.z := TO_LREAL(F_Merge24BitSigned(in[17], in[18], in[19]))*fRatioAcc;
END_METHOD

END_FUNCTION_BLOCK

// ---- IMU/POUs/FB_GetSerialData.TcPOU
FUNCTION_BLOCK FB_GetSerialData
VAR_INPUT
	bActive 			: BOOL := TRUE;
	// [in] Pointer to header
	pHeader 			: POINTER TO BYTE;
	// Size of header in bytes
	cbHeaderSize 		: UDINT;
	// Size of data packet in bytes (including header and checksum)
	cbPacketSize 		: UDINT;
	// [in] Reference to RxBuffer
	stRxBuffer 			: REFERENCE TO ComBuffer;
	// [out] Pointer to output data buffer
	pDataBuffer 		: POINTER TO BYTE;
	// Size of data packet in bytes
	cbDataBufferSize 	: UDINT;
END_VAR
VAR_OUTPUT
	// Number of discarded bytes due to lack of synchronisation
	nDiscardedBytes : UDINT := 0;
	// True if an error occured on last receive
	bError : BOOL;
	// Last error code (keeps last error code even if ther is no error, to check for error use bError)
	eLastError : E_SerialError;
	// Number of errors since startup
	nErrorCount : UDINT := 0;
	// Number of received (verified) datagrams per second
	nReceivedDatagrams : DINT := 0;
	// Number of dropped datagrams per second
	nDroppedDatagrams : DINT := 0;
END_VAR
VAR
	// True if a new unread data packet has been received
	bNewData : BOOL := FALSE;
	// State
	eSerialState : E_SerialState := E_SerialState.eStopped;
	// Buffer com, single byte
	fbReceiveByte : ReceiveByte;
	// Clears com buffer
	fbClearComBuffer : ClearComBuffer;
	// Timer
	fbTimer : TON := (PT := T#1S);
	// Received datagrams counter
	nReceivedCount : DINT := 0;
	// Dropped datagrams counter
	nDroppedCount : DINT := 0;
END_VAR

// Keep the com buffer cleared to avoid overflows when we are not active
IF NOT bActive THEN
	IF (stRxBuffer.Count > 0) THEN
		fbClearComBuffer(Buffer := stRxBuffer);
	END_IF
	
	eSerialState := E_SerialState.eStopped;
END_IF

IF (cbPacketSize > cbDataBufferSize) THEN
	bError := TRUE;
	eLastError := E_SerialError.eOutputBufferTooSmall;
ELSE
	bError := FALSE;
END_IF

fbTimer(IN := TRUE);
IF fbTimer.Q THEN
	fbTimer(IN := FALSE);
	nReceivedDatagrams := nReceivedCount;
	nReceivedCount := 0;
	nDroppedDatagrams := nDroppedCount;
	nDroppedCount := 0;
END_IF

CASE eSerialState OF
E_SerialState.eStopped:
	IF bActive THEN
		eSerialState := E_SerialState.eSearchForHeader;
	END_IF

E_SerialState.eSearchForHeader:
	searchForHeader(nMaxBytes := 100);
	
E_SerialState.eReceive:
	receive();

END_CASE

IF bError THEN
	nErrorCount := nErrorCount + 1;
END_IF

// Use this method to calculate checksum
// Returns true if the checksum is correct, false if it is incorrect
METHOD PRIVATE checksum : BOOL
VAR_INPUT
END_VAR
VAR CONSTANT
	ptSuffix : ARRAY [0..1] OF BYTE := [ 16#0D, 16#0A]; 
	crc_polynomial : UDINT := 16#04C11DB7;//16#82608EDB;//16#DB710641; //16#EDB88320;//16#04C11DB7;//divisor is 32bit 
	cbcrcSize : UDINT := 4;//Bytes
	cbsuffixLength: UDINT := 2;//Bytes
END_VAR
VAR
	calc_crc : UDINT := 0;//CRC value is 32bit
	received_crc : UDINT;
	i : UDINT ;
	j : UDINT ;
END_VAR

checksum := (pDataBuffer[63] = ptSuffix[0]) AND (pDataBuffer[64] = ptSuffix[1]);

IF NOT checksum THEN
	RETURN;
	
END_IF

//http://www.sunshine2k.de/articles/coding/crc/understanding_crc.html
calc_crc := 16#FFFFFFFF;
FOR i := 0 TO cbPacketSize-cbcrcSize-cbsuffixLength-1 DO
	calc_crc := calc_crc XOR SHL(TO_UDINT(pDataBuffer[i]),24); // move byte into MSB of 32bit CRC
	FOR j := 0 TO 7 DO 
		IF ((calc_crc AND 16#80000000) <> 0) THEN //test for MSB = bit 31
			calc_crc := (SHL(calc_crc,1) XOR crc_polynomial);
		ELSE 
			calc_crc := SHL(calc_crc,1); 
		END_IF		
	END_FOR
END_FOR

//We add one more byte added for normal datagram mode
calc_crc := calc_crc XOR 0; // move byte into MSB of 32bit CRC


FOR j := 0 TO 7 DO 
	IF ((calc_crc AND 16#80000000) <> 0) THEN //test for MSB = bit 31
		calc_crc := (SHL(calc_crc,1) XOR crc_polynomial);
	ELSE 
		calc_crc := SHL(calc_crc,1); 
	END_IF		
END_FOR

received_crc := SHL(TO_UDINT(pDataBuffer[59]), 24) OR SHL(TO_UDINT(pDataBuffer[60]), 16) OR SHL(TO_UDINT(pDataBuffer[61]), 8) OR TO_UDINT(pDataBuffer[62]);

checksum := calc_crc = received_crc;
END_METHOD

PROPERTY PUBLIC NewData : BOOL
GET
NewData := bNewData;
bNewData := FALSE;
END_GET
END_PROPERTY

METHOD PRIVATE receive
VAR_INPUT
END_VAR
VAR
	cbDataSize : UDINT;

	i : UDINT;
END_VAR
cbDataSize := (cbPacketSize - cbHeaderSize);

IF (stRxBuffer.Count < cbDataSize) THEN
	// Wait for more data
	RETURN;
END_IF

FOR i := 0 TO (cbDataSize - 1) DO
	fbReceiveByte(
		ReceivedByte => pDataBuffer[cbHeaderSize + i],
		RxBuffer := stRxBuffer
	);

	IF (fbReceiveByte.Error <> COMERROR_NOERROR) THEN
		bError := TRUE;
		eLastError := E_SerialError.eComBufferError;
		eSerialState := E_SerialState.eSearchForHeader;
		RETURN;
	END_IF
END_FOR

eSerialState := E_SerialState.eSearchForHeader;

IF NOT(checksum()) THEN
	bError := TRUE;
	eLastError := E_SerialError.eChecksumFailed;
	nDroppedCount := nDroppedCount + 1;
	RETURN;
END_IF

nDiscardedBytes := 0;
nReceivedCount := nReceivedCount + 1;
bNewData := TRUE;
END_METHOD

METHOD PRIVATE searchForHeader
VAR_INPUT
	// Set a maximum number of bytes to read each iteration in order to avoid getting stuck in an infinite loop
	nMaxBytes : UDINT;
END_VAR
VAR
	nBytesRead 	: UDINT;
	nHeaderByte : UDINT := 0;
	// nReceivedByte : BYTE;
END_VAR

FOR nBytesRead := 0 TO (nMaxBytes - 1) DO
	IF (stRxBuffer.Count < cbHeaderSize) THEN
		// Buffer content is less than the size of the header. Wait for more data
		RETURN;
	END_IF

	// Get a single byte from the buffer and compare to the header
	fbReceiveByte(
		ReceivedByte => pDataBuffer[nHeaderByte], // nReceivedByte,
		RxBuffer := stRxBuffer
	);
	
	IF (fbReceiveByte.Error <> COMERROR_NOERROR) THEN
		bError := TRUE;
		eLastError := E_SerialError.eComBufferError;
		EXIT;
	END_IF

	IF (pHeader[nHeaderByte] = pDataBuffer[nHeaderByte]) THEN
		// pDataBuffer[nHeaderByte] := nReceivedByte;
		nHeaderByte := nHeaderByte + 1;
	ELSE
		nDiscardedBytes := nDiscardedBytes + 1;
		nHeaderByte := 0;
	END_IF
	
	IF (nHeaderByte = cbHeaderSize) THEN
		// Header found :)
		eSerialState := E_SerialState.eReceive;
		// Run receive once in case we are already ready to read
		receive();
		EXIT;
	END_IF
END_FOR
END_METHOD

END_FUNCTION_BLOCK

// ---- IMU/POUs/FB_AccelerometerAngle.TcPOU
FUNCTION_BLOCK FB_AccelerometerAngle
VAR_INPUT
	fAx : LREAL;
	fAy : LREAL;
	fAz : LREAL;
END_VAR
VAR_OUTPUT
	fRoll 	: LREAL; // [rad]
	fPitch 	: LREAL; // [rad]
END_VAR
VAR
END_VAR

fRoll := ATAN2(fAy, fAz);

fPitch := ATAN2(-fAx, SQRT(EXPT(fAy, 2.0) + EXPT(fAz, 2.0)));

END_FUNCTION_BLOCK

// ---- IMU/POUs/ATAN2.TcPOU
FUNCTION ATAN2 : LREAL
VAR_INPUT
	y : LREAL;
	x : LREAL;
END_VAR
VAR
END_VAR

IF (x > 0.0) THEN
	// (x > 0)
	ATAN2 := 2*ATAN(y/(SQRT(EXPT(x, 2.0) + EXPT(y, 2.0)) + x));
ELSIF (y <> 0.0) THEN
	// (x <= 0) & (y != 0)
	ATAN2 := 2*ATAN((SQRT(EXPT(x, 2.0) + EXPT(y, 2.0)) - x)/y);
ELSIF (x < 0.0) THEN
	// (x < 0) & (y == 0)
	ATAN2 := PI;
ELSE
	// (x == 0) & (y == 0) Technically undefined, but we set it to zero
	ATAN2 := 0.0;
END_IF

END_FUNCTION

// ---- IMU/POUs/FB_ComplementaryFilter.TcPOU
FUNCTION_BLOCK FB_ComplementaryFilter
VAR_INPUT
	// Accelerometer angle [unit]
	fAccAngle 		: LREAL;
	// Gyro roll angle rate [unit/s]
	fGyroRate		: LREAL;
	// Filter ratio [0..1]
	fFilterRatio 	: LREAL;
	// Step time [s]
	fStepTime 		: LREAL;
END_VAR
VAR_OUTPUT
	// Filtered angle [unit]
	fAngle 	: LREAL := 0.0;
END_VAR
VAR
END_VAR


// θ(t) = (1 − α) · θ(t)a + α · (θt−1 + ω(t)g · dt)

fAngle := (1.0 - fFilterRatio)*fAccAngle + fFilterRatio*(fAngle + fGyroRate*fStepTime);

END_FUNCTION_BLOCK

// ---- POUs/F_Merge24BitSigned.TcPOU
FUNCTION F_Merge24BitSigned : DINT
VAR_INPUT
	byte_0 : BYTE;
	byte_1 : BYTE;
	byte_2 : BYTE;
END_VAR
VAR
	tmp : DWORD;
END_VAR


tmp := F_Merge24BitUnsigned(byte_0, byte_1, byte_2);

IF ((tmp AND 16#800000) <> 0) THEN // Check for sign bit
	// If signed then pad to invert 32 bit
	F_Merge24BitSigned := TO_DINT(tmp OR 16#FF000000);
ELSE
	// If unsigned then it's ok
	F_Merge24BitSigned := TO_DINT(tmp);
END_IF

END_FUNCTION

// ---- POUs/F_Merge24BitUnsigned.TcPOU
FUNCTION F_Merge24BitUnsigned : UDINT
VAR_INPUT
	byte_0 : BYTE;
	byte_1 : BYTE;
	byte_2 : BYTE;
END_VAR
VAR
END_VAR

F_Merge24BitUnsigned := SHL(TO_DWORD(byte_0) AND 16#FF, 16) OR SHL(TO_DWORD(byte_1) AND 16#FF, 8) OR TO_DWORD(byte_2) AND 16#FF;

END_FUNCTION
